	2://Prepear Write array befor write over ads
		//Standart Value
		//Type BOOL
		IF Lynus_Standards.GVL_Communicator.arrInterfaceInfoValueWriteTo[byReadWriteArrayNumber].sSymbolType = 'BOOL' AND TO_LWORD(Lynus_Standards.GVL_Communicator.arrInterfaceInfoValueWriteTo[byReadWriteArrayNumber].arrValue[1]) >= 0 AND TO_LWORD(Lynus_Standards.GVL_Communicator.arrInterfaceInfoValueWriteTo[byReadWriteArrayNumber].arrValue[1]) <= 1 THEN 
			arrBufferWrite_WriteAds[1] := STRING_TO_BYTE(Lynus_Standards.GVL_Communicator.arrInterfaceInfoValueWriteTo[byReadWriteArrayNumber].arrValue[1]); 
				bValueValid_WriteAds := TRUE;
					uiSizeToWrite_WriteAds := 1;
		END_IF
		//Type BYTE  	
		IF Lynus_Standards.GVL_Communicator.arrInterfaceInfoValueWriteTo[byReadWriteArrayNumber].sSymbolType = 'BYTE' AND TO_LWORD(Lynus_Standards.GVL_Communicator.arrInterfaceInfoValueWriteTo[byReadWriteArrayNumber].arrValue[1]) >= 0 AND TO_LWORD(Lynus_Standards.GVL_Communicator.arrInterfaceInfoValueWriteTo[byReadWriteArrayNumber].arrValue[1]) <= 255 THEN 
			arrBufferWrite_WriteAds[1] := STRING_TO_BYTE(Lynus_Standards.GVL_Communicator.arrInterfaceInfoValueWriteTo[byReadWriteArrayNumber].arrValue[1]); 
				bValueValid_WriteAds := TRUE;
					uiSizeToWrite_WriteAds := 1;
		END_IF
		//Type WORD
		IF Lynus_Standards.GVL_Communicator.arrInterfaceInfoValueWriteTo[byReadWriteArrayNumber].sSymbolType = 'WORD' AND TO_LWORD(Lynus_Standards.GVL_Communicator.arrInterfaceInfoValueWriteTo[byReadWriteArrayNumber].arrValue[1]) >= 0 AND TO_LWORD(Lynus_Standards.GVL_Communicator.arrInterfaceInfoValueWriteTo[byReadWriteArrayNumber].arrValue[1]) <= 65535 THEN 
			arrBufferWrite_WriteAds[2] := WORD_TO_BYTE(SHR(STRING_TO_WORD(Lynus_Standards.GVL_Communicator.arrInterfaceInfoValueWriteTo[byReadWriteArrayNumber].arrValue[1]),8) AND 16#FFFF);
			arrBufferWrite_WriteAds[1] := WORD_TO_BYTE(STRING_TO_WORD(Lynus_Standards.GVL_Communicator.arrInterfaceInfoValueWriteTo[byReadWriteArrayNumber].arrValue[1]) AND 16#FFFF); 
				bValueValid_WriteAds := TRUE;
					uiSizeToWrite_WriteAds := 2;
		END_IF
		//Type DWORD
		IF Lynus_Standards.GVL_Communicator.arrInterfaceInfoValueWriteTo[byReadWriteArrayNumber].sSymbolType = 'DWORD' AND TO_LWORD(Lynus_Standards.GVL_Communicator.arrInterfaceInfoValueWriteTo[byReadWriteArrayNumber].arrValue[1]) >= 0 AND TO_LWORD(Lynus_Standards.GVL_Communicator.arrInterfaceInfoValueWriteTo[byReadWriteArrayNumber].arrValue[1]) <= 4294967295 THEN 
			arrBufferWrite_WriteAds[4] := DWORD_TO_BYTE(SHR(STRING_TO_DWORD(Lynus_Standards.GVL_Communicator.arrInterfaceInfoValueWriteTo[byReadWriteArrayNumber].arrValue[1]),24) AND 16#FFFFFFFF);
			arrBufferWrite_WriteAds[3] := DWORD_TO_BYTE(SHR(STRING_TO_DWORD(Lynus_Standards.GVL_Communicator.arrInterfaceInfoValueWriteTo[byReadWriteArrayNumber].arrValue[1]),16) AND 16#FFFFFFFF);
			arrBufferWrite_WriteAds[2] := DWORD_TO_BYTE(SHR(STRING_TO_DWORD(Lynus_Standards.GVL_Communicator.arrInterfaceInfoValueWriteTo[byReadWriteArrayNumber].arrValue[1]),8) AND 16#FFFFFFFF);
			arrBufferWrite_WriteAds[1] := DWORD_TO_BYTE(STRING_TO_DWORD(Lynus_Standards.GVL_Communicator.arrInterfaceInfoValueWriteTo[byReadWriteArrayNumber].arrValue[1]) AND 16#FFFFFFFF); 
				bValueValid_WriteAds := TRUE;
					uiSizeToWrite_WriteAds := 4;
		END_IF
		//Type SINT
		IF Lynus_Standards.GVL_Communicator.arrInterfaceInfoValueWriteTo[byReadWriteArrayNumber].sSymbolType = 'SINT' AND TO_LINT(Lynus_Standards.GVL_Communicator.arrInterfaceInfoValueWriteTo[byReadWriteArrayNumber].arrValue[1]) >= -128 AND TO_LINT(Lynus_Standards.GVL_Communicator.arrInterfaceInfoValueWriteTo[byReadWriteArrayNumber].arrValue[1]) <= 127 THEN 
			arrBufferWrite_WriteAds[1] := SINT_TO_BYTE(STRING_TO_SINT(Lynus_Standards.GVL_Communicator.arrInterfaceInfoValueWriteTo[byReadWriteArrayNumber].arrValue[1])); 
				bValueValid_WriteAds := TRUE;
					uiSizeToWrite_WriteAds := 1;
		END_IF
		//Type USINT
		IF Lynus_Standards.GVL_Communicator.arrInterfaceInfoValueWriteTo[byReadWriteArrayNumber].sSymbolType = 'USINT' AND TO_LWORD(Lynus_Standards.GVL_Communicator.arrInterfaceInfoValueWriteTo[byReadWriteArrayNumber].arrValue[1]) >= 0 AND TO_LWORD(Lynus_Standards.GVL_Communicator.arrInterfaceInfoValueWriteTo[byReadWriteArrayNumber].arrValue[1]) <= 255 THEN 
			arrBufferWrite_WriteAds[1] := arrBufferWrite_WriteAds[1] := STRING_TO_USINT(Lynus_Standards.GVL_Communicator.arrInterfaceInfoValueWriteTo[byReadWriteArrayNumber].arrValue[1]); 
				bValueValid_WriteAds := TRUE;
					uiSizeToWrite_WriteAds := 1;
		END_IF
		//Type INT
		IF Lynus_Standards.GVL_Communicator.arrInterfaceInfoValueWriteTo[byReadWriteArrayNumber].sSymbolType = 'INT' AND TO_LINT(Lynus_Standards.GVL_Communicator.arrInterfaceInfoValueWriteTo[byReadWriteArrayNumber].arrValue[1]) >= -32768 AND TO_LINT(Lynus_Standards.GVL_Communicator.arrInterfaceInfoValueWriteTo[byReadWriteArrayNumber].arrValue[1]) <= 32767 THEN 
			arrBufferWrite_WriteAds[2] := UINT_TO_BYTE(SHR(INT_TO_UINT(STRING_TO_INT(Lynus_Standards.GVL_Communicator.arrInterfaceInfoValueWriteTo[byReadWriteArrayNumber].arrValue[1])),8) AND 16#FFFF);
			arrBufferWrite_WriteAds[1] := UINT_TO_BYTE(INT_TO_UINT(STRING_TO_INT(Lynus_Standards.GVL_Communicator.arrInterfaceInfoValueWriteTo[byReadWriteArrayNumber].arrValue[1])) AND 16#FFFF); 
				bValueValid_WriteAds := TRUE;
					uiSizeToWrite_WriteAds := 2;
		END_IF
		//Type UINT
		IF Lynus_Standards.GVL_Communicator.arrInterfaceInfoValueWriteTo[byReadWriteArrayNumber].sSymbolType = 'UINT' AND TO_LWORD(Lynus_Standards.GVL_Communicator.arrInterfaceInfoValueWriteTo[byReadWriteArrayNumber].arrValue[1]) >= 0 AND TO_LWORD(Lynus_Standards.GVL_Communicator.arrInterfaceInfoValueWriteTo[byReadWriteArrayNumber].arrValue[1]) <= 65535 THEN 
			arrBufferWrite_WriteAds[2] := UINT_TO_BYTE(SHR(STRING_TO_UINT(Lynus_Standards.GVL_Communicator.arrInterfaceInfoValueWriteTo[byReadWriteArrayNumber].arrValue[1]),8) AND 16#FFFF);
			arrBufferWrite_WriteAds[1] := UINT_TO_BYTE(STRING_TO_UINT(Lynus_Standards.GVL_Communicator.arrInterfaceInfoValueWriteTo[byReadWriteArrayNumber].arrValue[1]) AND 16#FFFF); 
				bValueValid_WriteAds := TRUE;
					uiSizeToWrite_WriteAds := 2;
		END_IF
		//Type DINT
		IF Lynus_Standards.GVL_Communicator.arrInterfaceInfoValueWriteTo[byReadWriteArrayNumber].sSymbolType = 'DINT' AND TO_LINT(Lynus_Standards.GVL_Communicator.arrInterfaceInfoValueWriteTo[byReadWriteArrayNumber].arrValue[1]) >= -2147483648 AND TO_LINT(Lynus_Standards.GVL_Communicator.arrInterfaceInfoValueWriteTo[byReadWriteArrayNumber].arrValue[1]) <= 2147483647 THEN 
			arrBufferWrite_WriteAds[4] := UDINT_TO_BYTE(SHR(DINT_TO_UDINT(STRING_TO_DINT(Lynus_Standards.GVL_Communicator.arrInterfaceInfoValueWriteTo[byReadWriteArrayNumber].arrValue[1])),24) AND 16#FFFFFFFF);
			arrBufferWrite_WriteAds[3] := UDINT_TO_BYTE(SHR(DINT_TO_UDINT(STRING_TO_DINT(Lynus_Standards.GVL_Communicator.arrInterfaceInfoValueWriteTo[byReadWriteArrayNumber].arrValue[1])),16) AND 16#FFFFFFFF);
			arrBufferWrite_WriteAds[2] := UDINT_TO_BYTE(SHR(DINT_TO_UDINT(STRING_TO_DINT(Lynus_Standards.GVL_Communicator.arrInterfaceInfoValueWriteTo[byReadWriteArrayNumber].arrValue[1])),8) AND 16#FFFFFFFF);
			arrBufferWrite_WriteAds[1] := UDINT_TO_BYTE(DINT_TO_UDINT(STRING_TO_DINT(Lynus_Standards.GVL_Communicator.arrInterfaceInfoValueWriteTo[byReadWriteArrayNumber].arrValue[1])) AND 16#FFFFFFF);
				bValueValid_WriteAds := TRUE;
					uiSizeToWrite_WriteAds := 4;
		END_IF
		//Type UDINT
		IF Lynus_Standards.GVL_Communicator.arrInterfaceInfoValueWriteTo[byReadWriteArrayNumber].sSymbolType = 'UDINT' AND TO_LWORD(Lynus_Standards.GVL_Communicator.arrInterfaceInfoValueWriteTo[byReadWriteArrayNumber].arrValue[1]) >= 0 AND TO_LWORD(Lynus_Standards.GVL_Communicator.arrInterfaceInfoValueWriteTo[byReadWriteArrayNumber].arrValue[1]) <= 4294967295 THEN 
			arrBufferWrite_WriteAds[4] := UDINT_TO_BYTE(SHR(STRING_TO_UDINT(Lynus_Standards.GVL_Communicator.arrInterfaceInfoValueWriteTo[byReadWriteArrayNumber].arrValue[1]),24) AND 16#FFFFFFFF);
			arrBufferWrite_WriteAds[3] := UDINT_TO_BYTE(SHR(STRING_TO_UDINT(Lynus_Standards.GVL_Communicator.arrInterfaceInfoValueWriteTo[byReadWriteArrayNumber].arrValue[1]),16) AND 16#FFFFFFFF);
			arrBufferWrite_WriteAds[2] := UDINT_TO_BYTE(SHR(STRING_TO_UDINT(Lynus_Standards.GVL_Communicator.arrInterfaceInfoValueWriteTo[byReadWriteArrayNumber].arrValue[1]),8) AND 16#FFFFFFFF);
			arrBufferWrite_WriteAds[1] := UDINT_TO_BYTE(STRING_TO_UDINT(Lynus_Standards.GVL_Communicator.arrInterfaceInfoValueWriteTo[byReadWriteArrayNumber].arrValue[1]) AND 16#FFFFFFFF); 
				bValueValid_WriteAds := TRUE;
					uiSizeToWrite_WriteAds := 4;
		END_IF
		//Type LINT
		IF Lynus_Standards.GVL_Communicator.arrInterfaceInfoValueWriteTo[byReadWriteArrayNumber].sSymbolType = 'LINT' AND TO_LINT(Lynus_Standards.GVL_Communicator.arrInterfaceInfoValueWriteTo[byReadWriteArrayNumber].arrValue[1]) >= -9223372036854775808 AND TO_LINT(Lynus_Standards.GVL_Communicator.arrInterfaceInfoValueWriteTo[byReadWriteArrayNumber].arrValue[1]) <= 9223372036854775807 THEN 
			arrBufferWrite_WriteAds[8] := ULINT_TO_BYTE(SHR(LINT_TO_ULINT(STRING_TO_LINT(Lynus_Standards.GVL_Communicator.arrInterfaceInfoValueWriteTo[byReadWriteArrayNumber].arrValue[1])),56) AND 16#FFFFFFFFFFFFFFFF);
			arrBufferWrite_WriteAds[7] := ULINT_TO_BYTE(SHR(LINT_TO_ULINT(STRING_TO_LINT(Lynus_Standards.GVL_Communicator.arrInterfaceInfoValueWriteTo[byReadWriteArrayNumber].arrValue[1])),48) AND 16#FFFFFFFFFFFFFFFF);
			arrBufferWrite_WriteAds[6] := ULINT_TO_BYTE(SHR(LINT_TO_ULINT(STRING_TO_LINT(Lynus_Standards.GVL_Communicator.arrInterfaceInfoValueWriteTo[byReadWriteArrayNumber].arrValue[1])),40) AND 16#FFFFFFFFFFFFFFFF);
			arrBufferWrite_WriteAds[5] := ULINT_TO_BYTE(SHR(LINT_TO_ULINT(STRING_TO_LINT(Lynus_Standards.GVL_Communicator.arrInterfaceInfoValueWriteTo[byReadWriteArrayNumber].arrValue[1])),32) AND 16#FFFFFFFFFFFFFFFF);
			arrBufferWrite_WriteAds[4] := ULINT_TO_BYTE(SHR(LINT_TO_ULINT(STRING_TO_LINT(Lynus_Standards.GVL_Communicator.arrInterfaceInfoValueWriteTo[byReadWriteArrayNumber].arrValue[1])),24) AND 16#FFFFFFFFFFFFFFFF);
			arrBufferWrite_WriteAds[3] := ULINT_TO_BYTE(SHR(LINT_TO_ULINT(STRING_TO_LINT(Lynus_Standards.GVL_Communicator.arrInterfaceInfoValueWriteTo[byReadWriteArrayNumber].arrValue[1])),16) AND 16#FFFFFFFFFFFFFFFF);
			arrBufferWrite_WriteAds[2] := ULINT_TO_BYTE(SHR(LINT_TO_ULINT(STRING_TO_LINT(Lynus_Standards.GVL_Communicator.arrInterfaceInfoValueWriteTo[byReadWriteArrayNumber].arrValue[1])),8) AND 16#FFFFFFFFFFFFFFFF);
			arrBufferWrite_WriteAds[1] := ULINT_TO_BYTE(LINT_TO_ULINT(STRING_TO_LINT(Lynus_Standards.GVL_Communicator.arrInterfaceInfoValueWriteTo[byReadWriteArrayNumber].arrValue[1])) AND 16#FFFFFFFFFFFFFFFF);
				bValueValid_WriteAds := TRUE;
					uiSizeToWrite_WriteAds := 8;
		END_IF
		//Type ULINT
		IF Lynus_Standards.GVL_Communicator.arrInterfaceInfoValueWriteTo[byReadWriteArrayNumber].sSymbolType = 'ULINT' AND TO_ULINT(Lynus_Standards.GVL_Communicator.arrInterfaceInfoValueWriteTo[byReadWriteArrayNumber].arrValue[1]) >= 0 AND TO_ULINT(Lynus_Standards.GVL_Communicator.arrInterfaceInfoValueWriteTo[byReadWriteArrayNumber].arrValue[1]) <= 18446744073709551615 THEN 
			arrBufferWrite_WriteAds[8] := ULINT_TO_BYTE(SHR(STRING_TO_ULINT(Lynus_Standards.GVL_Communicator.arrInterfaceInfoValueWriteTo[byReadWriteArrayNumber].arrValue[1]),56) AND 16#FFFFFFFFFFFFFFFF);
			arrBufferWrite_WriteAds[7] := ULINT_TO_BYTE(SHR(STRING_TO_ULINT(Lynus_Standards.GVL_Communicator.arrInterfaceInfoValueWriteTo[byReadWriteArrayNumber].arrValue[1]),48) AND 16#FFFFFFFFFFFFFFFF);
			arrBufferWrite_WriteAds[6] := ULINT_TO_BYTE(SHR(STRING_TO_ULINT(Lynus_Standards.GVL_Communicator.arrInterfaceInfoValueWriteTo[byReadWriteArrayNumber].arrValue[1]),40) AND 16#FFFFFFFFFFFFFFFF);
			arrBufferWrite_WriteAds[5] := ULINT_TO_BYTE(SHR(STRING_TO_ULINT(Lynus_Standards.GVL_Communicator.arrInterfaceInfoValueWriteTo[byReadWriteArrayNumber].arrValue[1]),32) AND 16#FFFFFFFFFFFFFFFF);
			arrBufferWrite_WriteAds[4] := ULINT_TO_BYTE(SHR(STRING_TO_ULINT(Lynus_Standards.GVL_Communicator.arrInterfaceInfoValueWriteTo[byReadWriteArrayNumber].arrValue[1]),24) AND 16#FFFFFFFFFFFFFFFF);
			arrBufferWrite_WriteAds[3] := ULINT_TO_BYTE(SHR(STRING_TO_ULINT(Lynus_Standards.GVL_Communicator.arrInterfaceInfoValueWriteTo[byReadWriteArrayNumber].arrValue[1]),16) AND 16#FFFFFFFFFFFFFFFF);
			arrBufferWrite_WriteAds[2] := ULINT_TO_BYTE(SHR(STRING_TO_ULINT(Lynus_Standards.GVL_Communicator.arrInterfaceInfoValueWriteTo[byReadWriteArrayNumber].arrValue[1]),8) AND 16#FFFFFFFFFFFFFFFF);
			arrBufferWrite_WriteAds[1] := ULINT_TO_BYTE(STRING_TO_ULINT(Lynus_Standards.GVL_Communicator.arrInterfaceInfoValueWriteTo[byReadWriteArrayNumber].arrValue[1]) AND 16#FFFFFFFFFFFFFFFF);
				bValueValid_WriteAds := TRUE;
					uiSizeToWrite_WriteAds := 8;
		END_IF
		//Type LWORD
		IF Lynus_Standards.GVL_Communicator.arrInterfaceInfoValueWriteTo[byReadWriteArrayNumber].sSymbolType = 'LWORD' AND TO_LWORD(Lynus_Standards.GVL_Communicator.arrInterfaceInfoValueWriteTo[byReadWriteArrayNumber].arrValue[1]) >= 0 AND TO_LWORD(Lynus_Standards.GVL_Communicator.arrInterfaceInfoValueWriteTo[byReadWriteArrayNumber].arrValue[1]) <= 18446744073709551615 THEN 
			arrBufferWrite_WriteAds[8] := LWORD_TO_BYTE(SHR(STRING_TO_LWORD(Lynus_Standards.GVL_Communicator.arrInterfaceInfoValueWriteTo[byReadWriteArrayNumber].arrValue[1]),56) AND 16#FFFFFFFFFFFFFFFF);
			arrBufferWrite_WriteAds[7] := LWORD_TO_BYTE(SHR(STRING_TO_LWORD(Lynus_Standards.GVL_Communicator.arrInterfaceInfoValueWriteTo[byReadWriteArrayNumber].arrValue[1]),48) AND 16#FFFFFFFFFFFFFFFF);
			arrBufferWrite_WriteAds[6] := LWORD_TO_BYTE(SHR(STRING_TO_LWORD(Lynus_Standards.GVL_Communicator.arrInterfaceInfoValueWriteTo[byReadWriteArrayNumber].arrValue[1]),40) AND 16#FFFFFFFFFFFFFFFF);
			arrBufferWrite_WriteAds[5] := LWORD_TO_BYTE(SHR(STRING_TO_LWORD(Lynus_Standards.GVL_Communicator.arrInterfaceInfoValueWriteTo[byReadWriteArrayNumber].arrValue[1]),32) AND 16#FFFFFFFFFFFFFFFF);
			arrBufferWrite_WriteAds[4] := LWORD_TO_BYTE(SHR(STRING_TO_LWORD(Lynus_Standards.GVL_Communicator.arrInterfaceInfoValueWriteTo[byReadWriteArrayNumber].arrValue[1]),24) AND 16#FFFFFFFFFFFFFFFF);
			arrBufferWrite_WriteAds[3] := LWORD_TO_BYTE(SHR(STRING_TO_LWORD(Lynus_Standards.GVL_Communicator.arrInterfaceInfoValueWriteTo[byReadWriteArrayNumber].arrValue[1]),16) AND 16#FFFFFFFFFFFFFFFF);
			arrBufferWrite_WriteAds[2] := LWORD_TO_BYTE(SHR(STRING_TO_LWORD(Lynus_Standards.GVL_Communicator.arrInterfaceInfoValueWriteTo[byReadWriteArrayNumber].arrValue[1]),8) AND 16#FFFFFFFFFFFFFFFF);
			arrBufferWrite_WriteAds[1] := LWORD_TO_BYTE(STRING_TO_LWORD(Lynus_Standards.GVL_Communicator.arrInterfaceInfoValueWriteTo[byReadWriteArrayNumber].arrValue[1]) AND 16#FFFFFFFFFFFFFFFF);
				bValueValid_WriteAds := TRUE;
					uiSizeToWrite_WriteAds := 8;
		END_IF
		//Type REAL
		IF Lynus_Standards.GVL_Communicator.arrInterfaceInfoValueWriteTo[byReadWriteArrayNumber].sSymbolType = 'REAL' AND LEN(Lynus_Standards.GVL_Communicator.arrInterfaceInfoValueWriteTo[byReadWriteArrayNumber].arrValue[1]) <= 30 AND TO_LREAL(Lynus_Standards.GVL_Communicator.arrInterfaceInfoValueWriteTo[byReadWriteArrayNumber].arrValue[1]) >= -3.40282326E+38 AND TO_LREAL(Lynus_Standards.GVL_Communicator.arrInterfaceInfoValueWriteTo[byReadWriteArrayNumber].arrValue[1]) <= 3.40282326E+38 THEN
			rRealValueCheckBeforWrite_WriteAds := STRING_TO_REAL(Lynus_Standards.GVL_Communicator.arrInterfaceInfoValueWriteTo[byReadWriteArrayNumber].arrValue[1]);
				IF IsFinite(F_REAL(rRealValueCheckBeforWrite_WriteAds)) THEN
					unConvertDWORD_TO_REAL_WriteAds.rValueFloat := STRING_TO_REAL(Lynus_Standards.GVL_Communicator.arrInterfaceInfoValueWriteTo[byReadWriteArrayNumber].arrValue[1]);
						arrBufferWrite_WriteAds[4] := UDINT_TO_BYTE((SHR(DWORD_TO_UDINT(unConvertDWORD_TO_REAL_WriteAds.dwRawValue),24) AND 16#FFFFFFFF));
						arrBufferWrite_WriteAds[3] := UDINT_TO_BYTE((SHR(DWORD_TO_UDINT(unConvertDWORD_TO_REAL_WriteAds.dwRawValue),16) AND 16#FFFFFFFF));
						arrBufferWrite_WriteAds[2] := UDINT_TO_BYTE((SHR(DWORD_TO_UDINT(unConvertDWORD_TO_REAL_WriteAds.dwRawValue),8) AND 16#FFFFFFFF));
						arrBufferWrite_WriteAds[1] := UDINT_TO_BYTE(DWORD_TO_UDINT(unConvertDWORD_TO_REAL_WriteAds.dwRawValue) AND 16#FFFFFFFF);
							bValueValid_WriteAds := TRUE;
								uiSizeToWrite_WriteAds := 4;
				END_IF					
		END_IF	
		//Type LREAL
		IF Lynus_Standards.GVL_Communicator.arrInterfaceInfoValueWriteTo[byReadWriteArrayNumber].sSymbolType = 'LREAL' AND LEN(Lynus_Standards.GVL_Communicator.arrInterfaceInfoValueWriteTo[byReadWriteArrayNumber].arrValue[1]) <= 30 AND TO_LREAL(Lynus_Standards.GVL_Communicator.arrInterfaceInfoValueWriteTo[byReadWriteArrayNumber].arrValue[1]) >= -1.7976931348623157E+307 AND TO_LREAL(Lynus_Standards.GVL_Communicator.arrInterfaceInfoValueWriteTo[byReadWriteArrayNumber].arrValue[1]) <= 1.7976931348623157E+307 THEN
			lrRealValueCheckBeforWrite_WriteAds := STRING_TO_LREAL(Lynus_Standards.GVL_Communicator.arrInterfaceInfoValueWriteTo[byReadWriteArrayNumber].arrValue[1]);
				IF IsFinite(F_LREAL(lrRealValueCheckBeforWrite_WriteAds)) THEN
					unConvertULINT_TO_LREAL_WriteAds.lrValueFloat := STRING_TO_LREAL(Lynus_Standards.GVL_Communicator.arrInterfaceInfoValueWriteTo[byReadWriteArrayNumber].arrValue[1]);
						arrBufferWrite_WriteAds[8] := LWORD_TO_BYTE((SHR(ULINT_TO_LWORD(unConvertULINT_TO_LREAL_WriteAds.uliRawValue),56) AND 16#FFFFFFFFFFFFFFFF));
						arrBufferWrite_WriteAds[7] := LWORD_TO_BYTE((SHR(ULINT_TO_LWORD(unConvertULINT_TO_LREAL_WriteAds.uliRawValue),48) AND 16#FFFFFFFFFFFFFFFF));
						arrBufferWrite_WriteAds[6] := LWORD_TO_BYTE((SHR(ULINT_TO_LWORD(unConvertULINT_TO_LREAL_WriteAds.uliRawValue),40) AND 16#FFFFFFFFFFFFFFFF));
						arrBufferWrite_WriteAds[5] := LWORD_TO_BYTE((SHR(ULINT_TO_LWORD(unConvertULINT_TO_LREAL_WriteAds.uliRawValue),32) AND 16#FFFFFFFFFFFFFFFF));
						arrBufferWrite_WriteAds[4] := LWORD_TO_BYTE((SHR(ULINT_TO_LWORD(unConvertULINT_TO_LREAL_WriteAds.uliRawValue),24) AND 16#FFFFFFFFFFFFFFFF));
						arrBufferWrite_WriteAds[3] := LWORD_TO_BYTE((SHR(ULINT_TO_LWORD(unConvertULINT_TO_LREAL_WriteAds.uliRawValue),16) AND 16#FFFFFFFFFFFFFFFF));
						arrBufferWrite_WriteAds[2] := LWORD_TO_BYTE((SHR(ULINT_TO_LWORD(unConvertULINT_TO_LREAL_WriteAds.uliRawValue),8) AND 16#FFFFFFFFFFFFFFFF));
						arrBufferWrite_WriteAds[1] := LWORD_TO_BYTE(ULINT_TO_LWORD(unConvertULINT_TO_LREAL_WriteAds.uliRawValue) AND 16#FFFFFFFFFFFFFFFF);
							bValueValid_WriteAds := TRUE;
								uiSizeToWrite_WriteAds := 8;
				END_IF
		END_IF
		//Type STRING(30)
		IF Lynus_Standards.GVL_Communicator.arrInterfaceInfoValueWriteTo[byReadWriteArrayNumber].sSymbolType = 'STRING(30)' AND LEN(Lynus_Standards.GVL_Communicator.arrInterfaceInfoValueWriteTo[byReadWriteArrayNumber].arrValue[1]) <= 30 AND FIND(Lynus_Standards.GVL_Communicator.arrInterfaceInfoValueWriteTo[byReadWriteArrayNumber].arrValue[1],'#EMPTY#') = 0 THEN 
			FOR byLPEncodeReceivedString_WriteAds := 1 TO 30 BY 1 DO 
				byCounterEncodeString_WriteAds := byCounterEncodeString_WriteAds + 1;
					byCounterEncodeString_WriteAds := LIMIT(1,byCounterEncodeString_WriteAds,30);
						arrBufferWrite_WriteAds[byCounterEncodeString_WriteAds] := F_ToASC(MID(Lynus_Standards.GVL_Communicator.arrInterfaceInfoValueWriteTo[byReadWriteArrayNumber].arrValue[1],1,byCounterEncodeString_WriteAds));
							bValueValid_WriteAds := TRUE;
								uiSizeToWrite_WriteAds := byCounterEncodeString_WriteAds + 1;
			END_FOR
		END_IF
		IF Lynus_Standards.GVL_Communicator.arrInterfaceInfoValueWriteTo[byReadWriteArrayNumber].sSymbolType = 'STRING(30)' AND LEN(Lynus_Standards.GVL_Communicator.arrInterfaceInfoValueWriteTo[byReadWriteArrayNumber].arrValue[1]) <= 30 AND FIND(Lynus_Standards.GVL_Communicator.arrInterfaceInfoValueWriteTo[byReadWriteArrayNumber].arrValue[1],'#EMPTY#') <> 0 THEN
			FOR byLPEncodeReceivedString_WriteAds := 1 TO 30 BY 1 DO 
				byCounterEncodeString_WriteAds := byCounterEncodeString_WriteAds + 1;
					byCounterEncodeString_WriteAds := LIMIT(1,byCounterEncodeString_WriteAds,30);
						arrBufferWrite_WriteAds[byCounterEncodeString_WriteAds] := F_ToASC('');
							bValueValid_WriteAds := TRUE;
								uiSizeToWrite_WriteAds := byCounterEncodeString_WriteAds + 1;
			END_FOR
		END_IF
		//Type TIME and TIME_OF_DAY
		IF ((Lynus_Standards.GVL_Communicator.arrInterfaceInfoValueWriteTo[byReadWriteArrayNumber].sSymbolType = 'TIME' OR Lynus_Standards.GVL_Communicator.arrInterfaceInfoValueWriteTo[byReadWriteArrayNumber].sSymbolType = 'TIME_OF_DAY') AND TO_LWORD(Lynus_Standards.GVL_Communicator.arrInterfaceInfoValueWriteTo[byReadWriteArrayNumber].arrValue[1]) >= 0 AND TO_LWORD(Lynus_Standards.GVL_Communicator.arrInterfaceInfoValueWriteTo[byReadWriteArrayNumber].arrValue[1]) <= 4294967295) THEN 
			arrBufferWrite_WriteAds[4] := UDINT_TO_BYTE(SHR(STRING_TO_UDINT(Lynus_Standards.GVL_Communicator.arrInterfaceInfoValueWriteTo[byReadWriteArrayNumber].arrValue[1]),24) AND 16#FFFFFFFF);
			arrBufferWrite_WriteAds[3] := UDINT_TO_BYTE(SHR(STRING_TO_UDINT(Lynus_Standards.GVL_Communicator.arrInterfaceInfoValueWriteTo[byReadWriteArrayNumber].arrValue[1]),16) AND 16#FFFFFFFF);
			arrBufferWrite_WriteAds[2] := UDINT_TO_BYTE(SHR(STRING_TO_UDINT(Lynus_Standards.GVL_Communicator.arrInterfaceInfoValueWriteTo[byReadWriteArrayNumber].arrValue[1]),8) AND 16#FFFFFFFF);
			arrBufferWrite_WriteAds[1] := UDINT_TO_BYTE(STRING_TO_UDINT(Lynus_Standards.GVL_Communicator.arrInterfaceInfoValueWriteTo[byReadWriteArrayNumber].arrValue[1]) AND 16#FFFFFFFF); 
				bValueValid_WriteAds := TRUE;
					uiSizeToWrite_WriteAds := 4;
		END_IF
		//Type DATE and DATE_AND_TIME
		IF ((Lynus_Standards.GVL_Communicator.arrInterfaceInfoValueWriteTo[byReadWriteArrayNumber].sSymbolType = 'DATE' OR Lynus_Standards.GVL_Communicator.arrInterfaceInfoValueWriteTo[byReadWriteArrayNumber].sSymbolType = 'DATE_AND_TIME') AND TO_LWORD(Lynus_Standards.GVL_Communicator.arrInterfaceInfoValueWriteTo[byReadWriteArrayNumber].arrValue[1]) >= 0 AND TO_LWORD(Lynus_Standards.GVL_Communicator.arrInterfaceInfoValueWriteTo[byReadWriteArrayNumber].arrValue[1]) <= 4294967295000) THEN 
			uliDate_WriteAds := STRING_TO_ULINT(Lynus_Standards.GVL_Communicator.arrInterfaceInfoValueWriteTo[byReadWriteArrayNumber].arrValue[1]);
				udiDate_WriteAds := ULINT_TO_UDINT(uliDate_WriteAds / 1000);	
					arrBufferWrite_WriteAds[4] := UDINT_TO_BYTE(SHR(udiDate_WriteAds,24) AND 16#FFFFFFFF);
					arrBufferWrite_WriteAds[3] := UDINT_TO_BYTE(SHR(udiDate_WriteAds,16) AND 16#FFFFFFFF);
					arrBufferWrite_WriteAds[2] := UDINT_TO_BYTE(SHR(udiDate_WriteAds,8) AND 16#FFFFFFFF);
					arrBufferWrite_WriteAds[1] := UDINT_TO_BYTE(udiDate_WriteAds AND 16#FFFFFFFF); 
						bValueValid_WriteAds := TRUE;
							uiSizeToWrite_WriteAds := 4;
		END_IF
			//Array with Standart Value
			//Type BOOL
			IF Lynus_Standards.GVL_Communicator.arrInterfaceInfoValueWriteTo[byReadWriteArrayNumber].uiSizeArray <= Lynus_Standards.Constants_Communicator.bySizeOfValueArray AND FIND(Lynus_Standards.GVL_Communicator.arrInterfaceInfoValueWriteTo[byReadWriteArrayNumber].sSymbolType,'OF BOOL') <> 0 THEN
				FOR uiLPWriteValueFromArray_WriteAds := 1 TO Lynus_Standards.GVL_Communicator.arrInterfaceInfoValueWriteTo[byReadWriteArrayNumber].uiSizeArray BY 1 DO
					IF TO_LWORD(Lynus_Standards.GVL_Communicator.arrInterfaceInfoValueWriteTo[byReadWriteArrayNumber].arrValue[uiLPWriteValueFromArray_WriteAds]) >= 0 AND TO_LWORD(Lynus_Standards.GVL_Communicator.arrInterfaceInfoValueWriteTo[byReadWriteArrayNumber].arrValue[uiLPWriteValueFromArray_WriteAds]) <= 1 THEN   
						arrBufferWrite_WriteAds[uiLPWriteValueFromArray_WriteAds] := STRING_TO_BYTE(Lynus_Standards.GVL_Communicator.arrInterfaceInfoValueWriteTo[byReadWriteArrayNumber].arrValue[uiLPWriteValueFromArray_WriteAds]); 
							uiSizeToWrite_WriteAds := 1 * Lynus_Standards.GVL_Communicator.arrInterfaceInfoValueWriteTo[byReadWriteArrayNumber].uiSizeArray;
								byCounterReceivedValueOK_WriteAds := byCounterReceivedValueOK_WriteAds + 1;
									byCounterReceivedValueOK_WriteAds := LIMIT(0,byCounterReceivedValueOK_WriteAds,Lynus_Standards.Constants_Communicator.bySizeOfValueArray);
										IF byCounterReceivedValueOK_WriteAds >= Lynus_Standards.GVL_Communicator.arrInterfaceInfoValueWriteTo[byReadWriteArrayNumber].uiSizeArray THEN bValueValid_WriteAds := TRUE; END_IF 
					END_IF
				END_FOR
			END_IF
			//Type BYTE
			IF Lynus_Standards.GVL_Communicator.arrInterfaceInfoValueWriteTo[byReadWriteArrayNumber].uiSizeArray <= Lynus_Standards.Constants_Communicator.bySizeOfValueArray AND FIND(Lynus_Standards.GVL_Communicator.arrInterfaceInfoValueWriteTo[byReadWriteArrayNumber].sSymbolType,'OF BYTE') <> 0 THEN
				FOR uiLPWriteValueFromArray_WriteAds := 1 TO Lynus_Standards.GVL_Communicator.arrInterfaceInfoValueWriteTo[byReadWriteArrayNumber].uiSizeArray BY 1 DO   
					IF TO_LWORD(Lynus_Standards.GVL_Communicator.arrInterfaceInfoValueWriteTo[byReadWriteArrayNumber].arrValue[uiLPWriteValueFromArray_WriteAds]) >= 0 AND TO_LWORD(Lynus_Standards.GVL_Communicator.arrInterfaceInfoValueWriteTo[byReadWriteArrayNumber].arrValue[uiLPWriteValueFromArray_WriteAds]) <= 255 THEN 
						arrBufferWrite_WriteAds[uiLPWriteValueFromArray_WriteAds] := STRING_TO_BYTE(Lynus_Standards.GVL_Communicator.arrInterfaceInfoValueWriteTo[byReadWriteArrayNumber].arrValue[uiLPWriteValueFromArray_WriteAds]); 
							uiSizeToWrite_WriteAds := 1 * Lynus_Standards.GVL_Communicator.arrInterfaceInfoValueWriteTo[byReadWriteArrayNumber].uiSizeArray;
								byCounterReceivedValueOK_WriteAds := byCounterReceivedValueOK_WriteAds + 1;
									byCounterReceivedValueOK_WriteAds := LIMIT(0,byCounterReceivedValueOK_WriteAds,Lynus_Standards.Constants_Communicator.bySizeOfValueArray);
										IF byCounterReceivedValueOK_WriteAds >= Lynus_Standards.GVL_Communicator.arrInterfaceInfoValueWriteTo[byReadWriteArrayNumber].uiSizeArray THEN bValueValid_WriteAds := TRUE; END_IF  
					END_IF
				END_FOR
			END_IF
			//Type WORD
			IF Lynus_Standards.GVL_Communicator.arrInterfaceInfoValueWriteTo[byReadWriteArrayNumber].uiSizeArray <= Lynus_Standards.Constants_Communicator.bySizeOfValueArray AND FIND(Lynus_Standards.GVL_Communicator.arrInterfaceInfoValueWriteTo[byReadWriteArrayNumber].sSymbolType,'OF WORD') <> 0 THEN
				FOR uiLPWriteValueFromArray_WriteAds := 1 TO Lynus_Standards.GVL_Communicator.arrInterfaceInfoValueWriteTo[byReadWriteArrayNumber].uiSizeArray BY 1 DO  
					IF TO_LWORD(Lynus_Standards.GVL_Communicator.arrInterfaceInfoValueWriteTo[byReadWriteArrayNumber].arrValue[uiLPWriteValueFromArray_WriteAds]) >= 0 AND TO_LWORD(Lynus_Standards.GVL_Communicator.arrInterfaceInfoValueWriteTo[byReadWriteArrayNumber].arrValue[uiLPWriteValueFromArray_WriteAds]) <= 65535 THEN  
						arrCounterWriteValueInArray_WriteAds[1] := LIMIT(1,arrCounterWriteValueInArray_WriteAds[1],2000); arrCounterWriteValueInArray_WriteAds[2] := LIMIT(2,arrCounterWriteValueInArray_WriteAds[2],2000);	
							arrBufferWrite_WriteAds[arrCounterWriteValueInArray_WriteAds[2]] := WORD_TO_BYTE(SHR(STRING_TO_WORD(Lynus_Standards.GVL_Communicator.arrInterfaceInfoValueWriteTo[byReadWriteArrayNumber].arrValue[uiLPWriteValueFromArray_WriteAds]),8) AND 16#FFFF);
							arrBufferWrite_WriteAds[arrCounterWriteValueInArray_WriteAds[1]] := WORD_TO_BYTE(STRING_TO_WORD(Lynus_Standards.GVL_Communicator.arrInterfaceInfoValueWriteTo[byReadWriteArrayNumber].arrValue[uiLPWriteValueFromArray_WriteAds]) AND 16#FFFF); 
						arrCounterWriteValueInArray_WriteAds[1] := arrCounterWriteValueInArray_WriteAds[1] + 2; arrCounterWriteValueInArray_WriteAds[2] := arrCounterWriteValueInArray_WriteAds[2] + 2;
							uiSizeToWrite_WriteAds := 2 * Lynus_Standards.GVL_Communicator.arrInterfaceInfoValueWriteTo[byReadWriteArrayNumber].uiSizeArray;
								byCounterReceivedValueOK_WriteAds := byCounterReceivedValueOK_WriteAds + 1;
									byCounterReceivedValueOK_WriteAds := LIMIT(0,byCounterReceivedValueOK_WriteAds,Lynus_Standards.Constants_Communicator.bySizeOfValueArray);
										IF byCounterReceivedValueOK_WriteAds >= Lynus_Standards.GVL_Communicator.arrInterfaceInfoValueWriteTo[byReadWriteArrayNumber].uiSizeArray THEN bValueValid_WriteAds := TRUE; END_IF  
					END_IF
				END_FOR
			END_IF
			//Type DWORD
			IF Lynus_Standards.GVL_Communicator.arrInterfaceInfoValueWriteTo[byReadWriteArrayNumber].uiSizeArray <= Lynus_Standards.Constants_Communicator.bySizeOfValueArray AND FIND(Lynus_Standards.GVL_Communicator.arrInterfaceInfoValueWriteTo[byReadWriteArrayNumber].sSymbolType,'OF DWORD') <> 0 THEN
				FOR uiLPWriteValueFromArray_WriteAds := 1 TO Lynus_Standards.GVL_Communicator.arrInterfaceInfoValueWriteTo[byReadWriteArrayNumber].uiSizeArray BY 1 DO 
					IF TO_LWORD(Lynus_Standards.GVL_Communicator.arrInterfaceInfoValueWriteTo[byReadWriteArrayNumber].arrValue[uiLPWriteValueFromArray_WriteAds]) >= 0 AND TO_LWORD(Lynus_Standards.GVL_Communicator.arrInterfaceInfoValueWriteTo[byReadWriteArrayNumber].arrValue[uiLPWriteValueFromArray_WriteAds]) <= 4294967295 THEN   
						arrCounterWriteValueInArray_WriteAds[1] := LIMIT(1,arrCounterWriteValueInArray_WriteAds[1],2000); arrCounterWriteValueInArray_WriteAds[2] := LIMIT(2,arrCounterWriteValueInArray_WriteAds[2],2000);
							arrCounterWriteValueInArray_WriteAds[3] := LIMIT(3,arrCounterWriteValueInArray_WriteAds[3],2000); arrCounterWriteValueInArray_WriteAds[4] := LIMIT(4,arrCounterWriteValueInArray_WriteAds[4],2000);	
								arrBufferWrite_WriteAds[arrCounterWriteValueInArray_WriteAds[4]] := DWORD_TO_BYTE(SHR(STRING_TO_DWORD(Lynus_Standards.GVL_Communicator.arrInterfaceInfoValueWriteTo[byReadWriteArrayNumber].arrValue[uiLPWriteValueFromArray_WriteAds]),24) AND 16#FFFFFFFF);
								arrBufferWrite_WriteAds[arrCounterWriteValueInArray_WriteAds[3]] := DWORD_TO_BYTE(SHR(STRING_TO_DWORD(Lynus_Standards.GVL_Communicator.arrInterfaceInfoValueWriteTo[byReadWriteArrayNumber].arrValue[uiLPWriteValueFromArray_WriteAds]),16) AND 16#FFFFFFFF);
								arrBufferWrite_WriteAds[arrCounterWriteValueInArray_WriteAds[2]] := DWORD_TO_BYTE(SHR(STRING_TO_DWORD(Lynus_Standards.GVL_Communicator.arrInterfaceInfoValueWriteTo[byReadWriteArrayNumber].arrValue[uiLPWriteValueFromArray_WriteAds]),8) AND 16#FFFFFFFF);
								arrBufferWrite_WriteAds[arrCounterWriteValueInArray_WriteAds[1]] := DWORD_TO_BYTE(STRING_TO_DWORD(Lynus_Standards.GVL_Communicator.arrInterfaceInfoValueWriteTo[byReadWriteArrayNumber].arrValue[uiLPWriteValueFromArray_WriteAds]) AND 16#FFFFFFFF); 
						arrCounterWriteValueInArray_WriteAds[1] := arrCounterWriteValueInArray_WriteAds[1] + 4; arrCounterWriteValueInArray_WriteAds[2] := arrCounterWriteValueInArray_WriteAds[2] + 4;
							arrCounterWriteValueInArray_WriteAds[3] := arrCounterWriteValueInArray_WriteAds[3] + 4; arrCounterWriteValueInArray_WriteAds[4] := arrCounterWriteValueInArray_WriteAds[4] + 4;
								uiSizeToWrite_WriteAds := 4 * Lynus_Standards.GVL_Communicator.arrInterfaceInfoValueWriteTo[byReadWriteArrayNumber].uiSizeArray;	
									byCounterReceivedValueOK_WriteAds := byCounterReceivedValueOK_WriteAds + 1;
										byCounterReceivedValueOK_WriteAds := LIMIT(0,byCounterReceivedValueOK_WriteAds,Lynus_Standards.Constants_Communicator.bySizeOfValueArray);
											IF byCounterReceivedValueOK_WriteAds >= Lynus_Standards.GVL_Communicator.arrInterfaceInfoValueWriteTo[byReadWriteArrayNumber].uiSizeArray THEN bValueValid_WriteAds := TRUE; END_IF  
					END_IF
				END_FOR
			END_IF
			//Type SINT
			IF Lynus_Standards.GVL_Communicator.arrInterfaceInfoValueWriteTo[byReadWriteArrayNumber].uiSizeArray <= Lynus_Standards.Constants_Communicator.bySizeOfValueArray AND FIND(Lynus_Standards.GVL_Communicator.arrInterfaceInfoValueWriteTo[byReadWriteArrayNumber].sSymbolType,'OF USINT') <> 0 THEN
				FOR uiLPWriteValueFromArray_WriteAds := 1 TO Lynus_Standards.GVL_Communicator.arrInterfaceInfoValueWriteTo[byReadWriteArrayNumber].uiSizeArray BY 1 DO   
					IF TO_LINT(Lynus_Standards.GVL_Communicator.arrInterfaceInfoValueWriteTo[byReadWriteArrayNumber].arrValue[uiLPWriteValueFromArray_WriteAds]) >= -128 AND TO_LINT(Lynus_Standards.GVL_Communicator.arrInterfaceInfoValueWriteTo[byReadWriteArrayNumber].arrValue[uiLPWriteValueFromArray_WriteAds]) <= 127 THEN 
						arrBufferWrite_WriteAds[uiLPWriteValueFromArray_WriteAds] := SINT_TO_BYTE(STRING_TO_SINT(Lynus_Standards.GVL_Communicator.arrInterfaceInfoValueWriteTo[byReadWriteArrayNumber].arrValue[uiLPWriteValueFromArray_WriteAds])); 
							uiSizeToWrite_WriteAds := 1 * Lynus_Standards.GVL_Communicator.arrInterfaceInfoValueWriteTo[byReadWriteArrayNumber].uiSizeArray;
								byCounterReceivedValueOK_WriteAds := byCounterReceivedValueOK_WriteAds + 1;
									byCounterReceivedValueOK_WriteAds := LIMIT(0,byCounterReceivedValueOK_WriteAds,Lynus_Standards.Constants_Communicator.bySizeOfValueArray);
										IF byCounterReceivedValueOK_WriteAds >= Lynus_Standards.GVL_Communicator.arrInterfaceInfoValueWriteTo[byReadWriteArrayNumber].uiSizeArray THEN bValueValid_WriteAds := TRUE; END_IF  
					END_IF
				END_FOR
			END_IF
			//Type USINT
			IF Lynus_Standards.GVL_Communicator.arrInterfaceInfoValueWriteTo[byReadWriteArrayNumber].uiSizeArray <= Lynus_Standards.Constants_Communicator.bySizeOfValueArray AND FIND(Lynus_Standards.GVL_Communicator.arrInterfaceInfoValueWriteTo[byReadWriteArrayNumber].sSymbolType,'OF USINT') <> 0 THEN
				FOR uiLPWriteValueFromArray_WriteAds := 1 TO Lynus_Standards.GVL_Communicator.arrInterfaceInfoValueWriteTo[byReadWriteArrayNumber].uiSizeArray BY 1 DO   
					IF TO_LWORD(Lynus_Standards.GVL_Communicator.arrInterfaceInfoValueWriteTo[byReadWriteArrayNumber].arrValue[uiLPWriteValueFromArray_WriteAds]) >= 0 AND TO_LWORD(Lynus_Standards.GVL_Communicator.arrInterfaceInfoValueWriteTo[byReadWriteArrayNumber].arrValue[uiLPWriteValueFromArray_WriteAds]) <= 255 THEN 
						arrBufferWrite_WriteAds[uiLPWriteValueFromArray_WriteAds] := STRING_TO_USINT(Lynus_Standards.GVL_Communicator.arrInterfaceInfoValueWriteTo[byReadWriteArrayNumber].arrValue[uiLPWriteValueFromArray_WriteAds]); 
							uiSizeToWrite_WriteAds := 1 * Lynus_Standards.GVL_Communicator.arrInterfaceInfoValueWriteTo[byReadWriteArrayNumber].uiSizeArray;
								byCounterReceivedValueOK_WriteAds := byCounterReceivedValueOK_WriteAds + 1;
									byCounterReceivedValueOK_WriteAds := LIMIT(0,byCounterReceivedValueOK_WriteAds,Lynus_Standards.Constants_Communicator.bySizeOfValueArray);
										IF byCounterReceivedValueOK_WriteAds >= Lynus_Standards.GVL_Communicator.arrInterfaceInfoValueWriteTo[byReadWriteArrayNumber].uiSizeArray THEN bValueValid_WriteAds := TRUE; END_IF  
					END_IF
				END_FOR
			END_IF
			//Type INT
			IF Lynus_Standards.GVL_Communicator.arrInterfaceInfoValueWriteTo[byReadWriteArrayNumber].uiSizeArray <= Lynus_Standards.Constants_Communicator.bySizeOfValueArray AND FIND(Lynus_Standards.GVL_Communicator.arrInterfaceInfoValueWriteTo[byReadWriteArrayNumber].sSymbolType,'OF INT') <> 0 THEN
				FOR uiLPWriteValueFromArray_WriteAds := 1 TO Lynus_Standards.GVL_Communicator.arrInterfaceInfoValueWriteTo[byReadWriteArrayNumber].uiSizeArray BY 1 DO   
					IF TO_LINT(Lynus_Standards.GVL_Communicator.arrInterfaceInfoValueWriteTo[byReadWriteArrayNumber].arrValue[uiLPWriteValueFromArray_WriteAds]) >= -32768 AND TO_LINT(Lynus_Standards.GVL_Communicator.arrInterfaceInfoValueWriteTo[byReadWriteArrayNumber].arrValue[uiLPWriteValueFromArray_WriteAds]) <= 32767 THEN 
						arrCounterWriteValueInArray_WriteAds[1] := LIMIT(1,arrCounterWriteValueInArray_WriteAds[1],2000); arrCounterWriteValueInArray_WriteAds[2] := LIMIT(2,arrCounterWriteValueInArray_WriteAds[2],2000);	
							arrBufferWrite_WriteAds[arrCounterWriteValueInArray_WriteAds[2]] := UINT_TO_BYTE(SHR(INT_TO_UINT(STRING_TO_INT(Lynus_Standards.GVL_Communicator.arrInterfaceInfoValueWriteTo[byReadWriteArrayNumber].arrValue[uiLPWriteValueFromArray_WriteAds])),8) AND 16#FFFF);
							arrBufferWrite_WriteAds[arrCounterWriteValueInArray_WriteAds[1]] := UINT_TO_BYTE(INT_TO_UINT(STRING_TO_INT(Lynus_Standards.GVL_Communicator.arrInterfaceInfoValueWriteTo[byReadWriteArrayNumber].arrValue[uiLPWriteValueFromArray_WriteAds])) AND 16#FFFF); 
						arrCounterWriteValueInArray_WriteAds[1] := arrCounterWriteValueInArray_WriteAds[1] + 2; arrCounterWriteValueInArray_WriteAds[2] := arrCounterWriteValueInArray_WriteAds[2] + 2;
							uiSizeToWrite_WriteAds := 2 * Lynus_Standards.GVL_Communicator.arrInterfaceInfoValueWriteTo[byReadWriteArrayNumber].uiSizeArray;
								byCounterReceivedValueOK_WriteAds := byCounterReceivedValueOK_WriteAds + 1;
									byCounterReceivedValueOK_WriteAds := LIMIT(0,byCounterReceivedValueOK_WriteAds,Lynus_Standards.Constants_Communicator.bySizeOfValueArray);
										IF byCounterReceivedValueOK_WriteAds >= Lynus_Standards.GVL_Communicator.arrInterfaceInfoValueWriteTo[byReadWriteArrayNumber].uiSizeArray THEN bValueValid_WriteAds := TRUE; END_IF  
					END_IF
				END_FOR
			END_IF
			//Type UINT
			IF Lynus_Standards.GVL_Communicator.arrInterfaceInfoValueWriteTo[byReadWriteArrayNumber].uiSizeArray <= Lynus_Standards.Constants_Communicator.bySizeOfValueArray AND FIND(Lynus_Standards.GVL_Communicator.arrInterfaceInfoValueWriteTo[byReadWriteArrayNumber].sSymbolType,'OF UINT') <> 0 THEN
				FOR uiLPWriteValueFromArray_WriteAds := 1 TO Lynus_Standards.GVL_Communicator.arrInterfaceInfoValueWriteTo[byReadWriteArrayNumber].uiSizeArray BY 1 DO  
					IF TO_LWORD(Lynus_Standards.GVL_Communicator.arrInterfaceInfoValueWriteTo[byReadWriteArrayNumber].arrValue[uiLPWriteValueFromArray_WriteAds]) >= 0 AND TO_LWORD(Lynus_Standards.GVL_Communicator.arrInterfaceInfoValueWriteTo[byReadWriteArrayNumber].arrValue[uiLPWriteValueFromArray_WriteAds]) <= 65535 THEN  
						arrCounterWriteValueInArray_WriteAds[1] := LIMIT(1,arrCounterWriteValueInArray_WriteAds[1],2000); arrCounterWriteValueInArray_WriteAds[2] := LIMIT(2,arrCounterWriteValueInArray_WriteAds[2],2000);	
							arrBufferWrite_WriteAds[arrCounterWriteValueInArray_WriteAds[2]] := UINT_TO_BYTE(SHR(STRING_TO_UINT(Lynus_Standards.GVL_Communicator.arrInterfaceInfoValueWriteTo[byReadWriteArrayNumber].arrValue[uiLPWriteValueFromArray_WriteAds]),8) AND 16#FFFF);
							arrBufferWrite_WriteAds[arrCounterWriteValueInArray_WriteAds[1]] := UINT_TO_BYTE(STRING_TO_UINT(Lynus_Standards.GVL_Communicator.arrInterfaceInfoValueWriteTo[byReadWriteArrayNumber].arrValue[uiLPWriteValueFromArray_WriteAds]) AND 16#FFFF);  
						arrCounterWriteValueInArray_WriteAds[1] := arrCounterWriteValueInArray_WriteAds[1] + 2; arrCounterWriteValueInArray_WriteAds[2] := arrCounterWriteValueInArray_WriteAds[2] + 2;
							uiSizeToWrite_WriteAds := 2 * Lynus_Standards.GVL_Communicator.arrInterfaceInfoValueWriteTo[byReadWriteArrayNumber].uiSizeArray;
								byCounterReceivedValueOK_WriteAds := byCounterReceivedValueOK_WriteAds + 1;
									byCounterReceivedValueOK_WriteAds := LIMIT(0,byCounterReceivedValueOK_WriteAds,Lynus_Standards.Constants_Communicator.bySizeOfValueArray);
										IF byCounterReceivedValueOK_WriteAds >= Lynus_Standards.GVL_Communicator.arrInterfaceInfoValueWriteTo[byReadWriteArrayNumber].uiSizeArray THEN bValueValid_WriteAds := TRUE; END_IF  
					END_IF
				END_FOR
			END_IF
			//Type DINT
			IF Lynus_Standards.GVL_Communicator.arrInterfaceInfoValueWriteTo[byReadWriteArrayNumber].uiSizeArray <= Lynus_Standards.Constants_Communicator.bySizeOfValueArray AND FIND(Lynus_Standards.GVL_Communicator.arrInterfaceInfoValueWriteTo[byReadWriteArrayNumber].sSymbolType,'OF DINT') <> 0 THEN
				FOR uiLPWriteValueFromArray_WriteAds := 1 TO Lynus_Standards.GVL_Communicator.arrInterfaceInfoValueWriteTo[byReadWriteArrayNumber].uiSizeArray BY 1 DO 
					IF TO_LINT(Lynus_Standards.GVL_Communicator.arrInterfaceInfoValueWriteTo[byReadWriteArrayNumber].arrValue[uiLPWriteValueFromArray_WriteAds]) >= -2147483648 AND TO_LINT(Lynus_Standards.GVL_Communicator.arrInterfaceInfoValueWriteTo[byReadWriteArrayNumber].arrValue[uiLPWriteValueFromArray_WriteAds]) <= 2147483647 THEN   
						arrCounterWriteValueInArray_WriteAds[1] := LIMIT(1,arrCounterWriteValueInArray_WriteAds[1],2000); arrCounterWriteValueInArray_WriteAds[2] := LIMIT(2,arrCounterWriteValueInArray_WriteAds[2],2000);
							arrCounterWriteValueInArray_WriteAds[3] := LIMIT(3,arrCounterWriteValueInArray_WriteAds[3],2000); arrCounterWriteValueInArray_WriteAds[4] := LIMIT(4,arrCounterWriteValueInArray_WriteAds[4],2000);	
								arrBufferWrite_WriteAds[arrCounterWriteValueInArray_WriteAds[4]] := UDINT_TO_BYTE(SHR(DINT_TO_UDINT(STRING_TO_DINT(Lynus_Standards.GVL_Communicator.arrInterfaceInfoValueWriteTo[byReadWriteArrayNumber].arrValue[uiLPWriteValueFromArray_WriteAds])),24) AND 16#FFFFFFFF);
								arrBufferWrite_WriteAds[arrCounterWriteValueInArray_WriteAds[3]] := UDINT_TO_BYTE(SHR(DINT_TO_UDINT(STRING_TO_DINT(Lynus_Standards.GVL_Communicator.arrInterfaceInfoValueWriteTo[byReadWriteArrayNumber].arrValue[uiLPWriteValueFromArray_WriteAds])),16) AND 16#FFFFFFFF);
								arrBufferWrite_WriteAds[arrCounterWriteValueInArray_WriteAds[2]] := UDINT_TO_BYTE(SHR(DINT_TO_UDINT(STRING_TO_DINT(Lynus_Standards.GVL_Communicator.arrInterfaceInfoValueWriteTo[byReadWriteArrayNumber].arrValue[uiLPWriteValueFromArray_WriteAds])),8) AND 16#FFFFFFFF);
								arrBufferWrite_WriteAds[arrCounterWriteValueInArray_WriteAds[1]] := UDINT_TO_BYTE(DINT_TO_UDINT(STRING_TO_DINT(Lynus_Standards.GVL_Communicator.arrInterfaceInfoValueWriteTo[byReadWriteArrayNumber].arrValue[uiLPWriteValueFromArray_WriteAds])) AND 16#FFFFFFF); 
						arrCounterWriteValueInArray_WriteAds[1] := arrCounterWriteValueInArray_WriteAds[1] + 4; arrCounterWriteValueInArray_WriteAds[2] := arrCounterWriteValueInArray_WriteAds[2] + 4;
							arrCounterWriteValueInArray_WriteAds[3] := arrCounterWriteValueInArray_WriteAds[3] + 4; arrCounterWriteValueInArray_WriteAds[4] := arrCounterWriteValueInArray_WriteAds[4] + 4;
								uiSizeToWrite_WriteAds := 4 * Lynus_Standards.GVL_Communicator.arrInterfaceInfoValueWriteTo[byReadWriteArrayNumber].uiSizeArray;	
									byCounterReceivedValueOK_WriteAds := byCounterReceivedValueOK_WriteAds + 1;
										byCounterReceivedValueOK_WriteAds := LIMIT(0,byCounterReceivedValueOK_WriteAds,Lynus_Standards.Constants_Communicator.bySizeOfValueArray);
											IF byCounterReceivedValueOK_WriteAds >= Lynus_Standards.GVL_Communicator.arrInterfaceInfoValueWriteTo[byReadWriteArrayNumber].uiSizeArray THEN bValueValid_WriteAds := TRUE; END_IF  
					END_IF
				END_FOR
			END_IF
			//Type UDINT
			IF Lynus_Standards.GVL_Communicator.arrInterfaceInfoValueWriteTo[byReadWriteArrayNumber].uiSizeArray <= Lynus_Standards.Constants_Communicator.bySizeOfValueArray AND FIND(Lynus_Standards.GVL_Communicator.arrInterfaceInfoValueWriteTo[byReadWriteArrayNumber].sSymbolType,'OF UDINT') <> 0 THEN
				FOR uiLPWriteValueFromArray_WriteAds := 1 TO Lynus_Standards.GVL_Communicator.arrInterfaceInfoValueWriteTo[byReadWriteArrayNumber].uiSizeArray BY 1 DO 
					IF TO_LWORD(Lynus_Standards.GVL_Communicator.arrInterfaceInfoValueWriteTo[byReadWriteArrayNumber].arrValue[uiLPWriteValueFromArray_WriteAds]) >= 0 AND TO_LWORD(Lynus_Standards.GVL_Communicator.arrInterfaceInfoValueWriteTo[byReadWriteArrayNumber].arrValue[uiLPWriteValueFromArray_WriteAds]) <= 4294967295 THEN   
						arrCounterWriteValueInArray_WriteAds[1] := LIMIT(1,arrCounterWriteValueInArray_WriteAds[1],2000); arrCounterWriteValueInArray_WriteAds[2] := LIMIT(2,arrCounterWriteValueInArray_WriteAds[2],2000);
							arrCounterWriteValueInArray_WriteAds[3] := LIMIT(3,arrCounterWriteValueInArray_WriteAds[3],2000); arrCounterWriteValueInArray_WriteAds[4] := LIMIT(4,arrCounterWriteValueInArray_WriteAds[4],2000);	
								arrBufferWrite_WriteAds[arrCounterWriteValueInArray_WriteAds[4]] := UDINT_TO_BYTE(SHR(STRING_TO_UDINT(Lynus_Standards.GVL_Communicator.arrInterfaceInfoValueWriteTo[byReadWriteArrayNumber].arrValue[uiLPWriteValueFromArray_WriteAds]),24) AND 16#FFFFFFFF);
								arrBufferWrite_WriteAds[arrCounterWriteValueInArray_WriteAds[3]] := UDINT_TO_BYTE(SHR(STRING_TO_UDINT(Lynus_Standards.GVL_Communicator.arrInterfaceInfoValueWriteTo[byReadWriteArrayNumber].arrValue[uiLPWriteValueFromArray_WriteAds]),16) AND 16#FFFFFFFF);
								arrBufferWrite_WriteAds[arrCounterWriteValueInArray_WriteAds[2]] := UDINT_TO_BYTE(SHR(STRING_TO_UDINT(Lynus_Standards.GVL_Communicator.arrInterfaceInfoValueWriteTo[byReadWriteArrayNumber].arrValue[uiLPWriteValueFromArray_WriteAds]),8) AND 16#FFFFFFFF);
								arrBufferWrite_WriteAds[arrCounterWriteValueInArray_WriteAds[1]] := UDINT_TO_BYTE(STRING_TO_UDINT(Lynus_Standards.GVL_Communicator.arrInterfaceInfoValueWriteTo[byReadWriteArrayNumber].arrValue[uiLPWriteValueFromArray_WriteAds]) AND 16#FFFFFFFF);  
						arrCounterWriteValueInArray_WriteAds[1] := arrCounterWriteValueInArray_WriteAds[1] + 4; arrCounterWriteValueInArray_WriteAds[2] := arrCounterWriteValueInArray_WriteAds[2] + 4;
							arrCounterWriteValueInArray_WriteAds[3] := arrCounterWriteValueInArray_WriteAds[3] + 4; arrCounterWriteValueInArray_WriteAds[4] := arrCounterWriteValueInArray_WriteAds[4] + 4;
								uiSizeToWrite_WriteAds := 4 * Lynus_Standards.GVL_Communicator.arrInterfaceInfoValueWriteTo[byReadWriteArrayNumber].uiSizeArray;	
									byCounterReceivedValueOK_WriteAds := byCounterReceivedValueOK_WriteAds + 1;
										byCounterReceivedValueOK_WriteAds := LIMIT(0,byCounterReceivedValueOK_WriteAds,Lynus_Standards.Constants_Communicator.bySizeOfValueArray);
											IF byCounterReceivedValueOK_WriteAds >= Lynus_Standards.GVL_Communicator.arrInterfaceInfoValueWriteTo[byReadWriteArrayNumber].uiSizeArray THEN bValueValid_WriteAds := TRUE; END_IF  
					END_IF
				END_FOR
			END_IF
			//Type LINT
			IF Lynus_Standards.GVL_Communicator.arrInterfaceInfoValueWriteTo[byReadWriteArrayNumber].uiSizeArray <= Lynus_Standards.Constants_Communicator.bySizeOfValueArray AND FIND(Lynus_Standards.GVL_Communicator.arrInterfaceInfoValueWriteTo[byReadWriteArrayNumber].sSymbolType,'OF LINT') <> 0 THEN
				FOR uiLPWriteValueFromArray_WriteAds := 1 TO Lynus_Standards.GVL_Communicator.arrInterfaceInfoValueWriteTo[byReadWriteArrayNumber].uiSizeArray BY 1 DO 
					IF TO_LINT(Lynus_Standards.GVL_Communicator.arrInterfaceInfoValueWriteTo[byReadWriteArrayNumber].arrValue[uiLPWriteValueFromArray_WriteAds]) >= -9223372036854775808 AND TO_LINT(Lynus_Standards.GVL_Communicator.arrInterfaceInfoValueWriteTo[byReadWriteArrayNumber].arrValue[uiLPWriteValueFromArray_WriteAds]) <= 9223372036854775807 THEN   
						arrCounterWriteValueInArray_WriteAds[1] := LIMIT(1,arrCounterWriteValueInArray_WriteAds[1],2000); arrCounterWriteValueInArray_WriteAds[2] := LIMIT(2,arrCounterWriteValueInArray_WriteAds[2],2000);
							arrCounterWriteValueInArray_WriteAds[3] := LIMIT(3,arrCounterWriteValueInArray_WriteAds[3],2000); arrCounterWriteValueInArray_WriteAds[4] := LIMIT(4,arrCounterWriteValueInArray_WriteAds[4],2000);	
								arrCounterWriteValueInArray_WriteAds[5] := LIMIT(5,arrCounterWriteValueInArray_WriteAds[5],2000); arrCounterWriteValueInArray_WriteAds[6] := LIMIT(6,arrCounterWriteValueInArray_WriteAds[6],2000);
									arrCounterWriteValueInArray_WriteAds[7] := LIMIT(7,arrCounterWriteValueInArray_WriteAds[7],2000); arrCounterWriteValueInArray_WriteAds[8] := LIMIT(8,arrCounterWriteValueInArray_WriteAds[8],2000);	
										arrBufferWrite_WriteAds[arrCounterWriteValueInArray_WriteAds[8]] := ULINT_TO_BYTE(SHR(LINT_TO_ULINT(STRING_TO_LINT(Lynus_Standards.GVL_Communicator.arrInterfaceInfoValueWriteTo[byReadWriteArrayNumber].arrValue[uiLPWriteValueFromArray_WriteAds])),56) AND 16#FFFFFFFFFFFFFFFF);
										arrBufferWrite_WriteAds[arrCounterWriteValueInArray_WriteAds[7]] := ULINT_TO_BYTE(SHR(LINT_TO_ULINT(STRING_TO_LINT(Lynus_Standards.GVL_Communicator.arrInterfaceInfoValueWriteTo[byReadWriteArrayNumber].arrValue[uiLPWriteValueFromArray_WriteAds])),48) AND 16#FFFFFFFFFFFFFFFF);
										arrBufferWrite_WriteAds[arrCounterWriteValueInArray_WriteAds[6]] := ULINT_TO_BYTE(SHR(LINT_TO_ULINT(STRING_TO_LINT(Lynus_Standards.GVL_Communicator.arrInterfaceInfoValueWriteTo[byReadWriteArrayNumber].arrValue[uiLPWriteValueFromArray_WriteAds])),40) AND 16#FFFFFFFFFFFFFFFF);
										arrBufferWrite_WriteAds[arrCounterWriteValueInArray_WriteAds[5]] := ULINT_TO_BYTE(SHR(LINT_TO_ULINT(STRING_TO_LINT(Lynus_Standards.GVL_Communicator.arrInterfaceInfoValueWriteTo[byReadWriteArrayNumber].arrValue[uiLPWriteValueFromArray_WriteAds])),32) AND 16#FFFFFFFFFFFFFFFF);
										arrBufferWrite_WriteAds[arrCounterWriteValueInArray_WriteAds[4]] := ULINT_TO_BYTE(SHR(LINT_TO_ULINT(STRING_TO_LINT(Lynus_Standards.GVL_Communicator.arrInterfaceInfoValueWriteTo[byReadWriteArrayNumber].arrValue[uiLPWriteValueFromArray_WriteAds])),24) AND 16#FFFFFFFFFFFFFFFF);
										arrBufferWrite_WriteAds[arrCounterWriteValueInArray_WriteAds[3]] := ULINT_TO_BYTE(SHR(LINT_TO_ULINT(STRING_TO_LINT(Lynus_Standards.GVL_Communicator.arrInterfaceInfoValueWriteTo[byReadWriteArrayNumber].arrValue[uiLPWriteValueFromArray_WriteAds])),16) AND 16#FFFFFFFFFFFFFFFF);
										arrBufferWrite_WriteAds[arrCounterWriteValueInArray_WriteAds[2]] := ULINT_TO_BYTE(SHR(LINT_TO_ULINT(STRING_TO_LINT(Lynus_Standards.GVL_Communicator.arrInterfaceInfoValueWriteTo[byReadWriteArrayNumber].arrValue[uiLPWriteValueFromArray_WriteAds])),8) AND 16#FFFFFFFFFFFFFFFF);
										arrBufferWrite_WriteAds[arrCounterWriteValueInArray_WriteAds[1]] := ULINT_TO_BYTE(LINT_TO_ULINT(STRING_TO_LINT(Lynus_Standards.GVL_Communicator.arrInterfaceInfoValueWriteTo[byReadWriteArrayNumber].arrValue[uiLPWriteValueFromArray_WriteAds])) AND 16#FFFFFFFFFFFFFFFF);
						arrCounterWriteValueInArray_WriteAds[1] := arrCounterWriteValueInArray_WriteAds[1] + 8; arrCounterWriteValueInArray_WriteAds[2] := arrCounterWriteValueInArray_WriteAds[2] + 8;
							arrCounterWriteValueInArray_WriteAds[3] := arrCounterWriteValueInArray_WriteAds[3] + 8; arrCounterWriteValueInArray_WriteAds[4] := arrCounterWriteValueInArray_WriteAds[4] + 8;
								arrCounterWriteValueInArray_WriteAds[5] := arrCounterWriteValueInArray_WriteAds[5] + 8; arrCounterWriteValueInArray_WriteAds[6] := arrCounterWriteValueInArray_WriteAds[6] + 8;
									arrCounterWriteValueInArray_WriteAds[7] := arrCounterWriteValueInArray_WriteAds[7] + 8; arrCounterWriteValueInArray_WriteAds[8] := arrCounterWriteValueInArray_WriteAds[8] + 8;
										uiSizeToWrite_WriteAds := 8 * Lynus_Standards.GVL_Communicator.arrInterfaceInfoValueWriteTo[byReadWriteArrayNumber].uiSizeArray;	
											byCounterReceivedValueOK_WriteAds := byCounterReceivedValueOK_WriteAds + 1;
												byCounterReceivedValueOK_WriteAds := LIMIT(0,byCounterReceivedValueOK_WriteAds,Lynus_Standards.Constants_Communicator.bySizeOfValueArray);
													IF byCounterReceivedValueOK_WriteAds >= Lynus_Standards.GVL_Communicator.arrInterfaceInfoValueWriteTo[byReadWriteArrayNumber].uiSizeArray THEN bValueValid_WriteAds := TRUE; END_IF  
					END_IF
				END_FOR
			END_IF
			//Type ULINT
			IF Lynus_Standards.GVL_Communicator.arrInterfaceInfoValueWriteTo[byReadWriteArrayNumber].uiSizeArray <= Lynus_Standards.Constants_Communicator.bySizeOfValueArray AND FIND(Lynus_Standards.GVL_Communicator.arrInterfaceInfoValueWriteTo[byReadWriteArrayNumber].sSymbolType,'OF ULINT') <> 0 THEN
				FOR uiLPWriteValueFromArray_WriteAds := 1 TO Lynus_Standards.GVL_Communicator.arrInterfaceInfoValueWriteTo[byReadWriteArrayNumber].uiSizeArray BY 1 DO 
					IF TO_ULINT(Lynus_Standards.GVL_Communicator.arrInterfaceInfoValueWriteTo[byReadWriteArrayNumber].arrValue[uiLPWriteValueFromArray_WriteAds]) >= 0 AND TO_ULINT(Lynus_Standards.GVL_Communicator.arrInterfaceInfoValueWriteTo[byReadWriteArrayNumber].arrValue[uiLPWriteValueFromArray_WriteAds]) <= 18446744073709551615 THEN   
						arrCounterWriteValueInArray_WriteAds[1] := LIMIT(1,arrCounterWriteValueInArray_WriteAds[1],2000); arrCounterWriteValueInArray_WriteAds[2] := LIMIT(2,arrCounterWriteValueInArray_WriteAds[2],2000);
							arrCounterWriteValueInArray_WriteAds[3] := LIMIT(3,arrCounterWriteValueInArray_WriteAds[3],2000); arrCounterWriteValueInArray_WriteAds[4] := LIMIT(4,arrCounterWriteValueInArray_WriteAds[4],2000);	
								arrCounterWriteValueInArray_WriteAds[5] := LIMIT(5,arrCounterWriteValueInArray_WriteAds[5],2000); arrCounterWriteValueInArray_WriteAds[6] := LIMIT(6,arrCounterWriteValueInArray_WriteAds[6],2000);
									arrCounterWriteValueInArray_WriteAds[7] := LIMIT(7,arrCounterWriteValueInArray_WriteAds[7],2000); arrCounterWriteValueInArray_WriteAds[8] := LIMIT(8,arrCounterWriteValueInArray_WriteAds[8],2000);	
										arrBufferWrite_WriteAds[arrCounterWriteValueInArray_WriteAds[8]] := ULINT_TO_BYTE(SHR(STRING_TO_ULINT(Lynus_Standards.GVL_Communicator.arrInterfaceInfoValueWriteTo[byReadWriteArrayNumber].arrValue[uiLPWriteValueFromArray_WriteAds]),56) AND 16#FFFFFFFFFFFFFFFF);
										arrBufferWrite_WriteAds[arrCounterWriteValueInArray_WriteAds[7]] := ULINT_TO_BYTE(SHR(STRING_TO_ULINT(Lynus_Standards.GVL_Communicator.arrInterfaceInfoValueWriteTo[byReadWriteArrayNumber].arrValue[uiLPWriteValueFromArray_WriteAds]),48) AND 16#FFFFFFFFFFFFFFFF);
										arrBufferWrite_WriteAds[arrCounterWriteValueInArray_WriteAds[6]] := ULINT_TO_BYTE(SHR(STRING_TO_ULINT(Lynus_Standards.GVL_Communicator.arrInterfaceInfoValueWriteTo[byReadWriteArrayNumber].arrValue[uiLPWriteValueFromArray_WriteAds]),40) AND 16#FFFFFFFFFFFFFFFF);
										arrBufferWrite_WriteAds[arrCounterWriteValueInArray_WriteAds[5]] := ULINT_TO_BYTE(SHR(STRING_TO_ULINT(Lynus_Standards.GVL_Communicator.arrInterfaceInfoValueWriteTo[byReadWriteArrayNumber].arrValue[uiLPWriteValueFromArray_WriteAds]),32) AND 16#FFFFFFFFFFFFFFFF);
										arrBufferWrite_WriteAds[arrCounterWriteValueInArray_WriteAds[4]] := ULINT_TO_BYTE(SHR(STRING_TO_ULINT(Lynus_Standards.GVL_Communicator.arrInterfaceInfoValueWriteTo[byReadWriteArrayNumber].arrValue[uiLPWriteValueFromArray_WriteAds]),24) AND 16#FFFFFFFFFFFFFFFF);
										arrBufferWrite_WriteAds[arrCounterWriteValueInArray_WriteAds[3]] := ULINT_TO_BYTE(SHR(STRING_TO_ULINT(Lynus_Standards.GVL_Communicator.arrInterfaceInfoValueWriteTo[byReadWriteArrayNumber].arrValue[uiLPWriteValueFromArray_WriteAds]),16) AND 16#FFFFFFFFFFFFFFFF);
										arrBufferWrite_WriteAds[arrCounterWriteValueInArray_WriteAds[2]] := ULINT_TO_BYTE(SHR(STRING_TO_ULINT(Lynus_Standards.GVL_Communicator.arrInterfaceInfoValueWriteTo[byReadWriteArrayNumber].arrValue[uiLPWriteValueFromArray_WriteAds]),8) AND 16#FFFFFFFFFFFFFFFF);
										arrBufferWrite_WriteAds[arrCounterWriteValueInArray_WriteAds[1]] := ULINT_TO_BYTE(STRING_TO_ULINT(Lynus_Standards.GVL_Communicator.arrInterfaceInfoValueWriteTo[byReadWriteArrayNumber].arrValue[uiLPWriteValueFromArray_WriteAds]) AND 16#FFFFFFFFFFFFFFFF);
						arrCounterWriteValueInArray_WriteAds[1] := arrCounterWriteValueInArray_WriteAds[1] + 8; arrCounterWriteValueInArray_WriteAds[2] := arrCounterWriteValueInArray_WriteAds[2] + 8;
							arrCounterWriteValueInArray_WriteAds[3] := arrCounterWriteValueInArray_WriteAds[3] + 8; arrCounterWriteValueInArray_WriteAds[4] := arrCounterWriteValueInArray_WriteAds[4] + 8;
								arrCounterWriteValueInArray_WriteAds[5] := arrCounterWriteValueInArray_WriteAds[5] + 8; arrCounterWriteValueInArray_WriteAds[6] := arrCounterWriteValueInArray_WriteAds[6] + 8;
									arrCounterWriteValueInArray_WriteAds[7] := arrCounterWriteValueInArray_WriteAds[7] + 8; arrCounterWriteValueInArray_WriteAds[8] := arrCounterWriteValueInArray_WriteAds[8] + 8;
										uiSizeToWrite_WriteAds := 8 * Lynus_Standards.GVL_Communicator.arrInterfaceInfoValueWriteTo[byReadWriteArrayNumber].uiSizeArray;	
											byCounterReceivedValueOK_WriteAds := byCounterReceivedValueOK_WriteAds + 1;
												byCounterReceivedValueOK_WriteAds := LIMIT(0,byCounterReceivedValueOK_WriteAds,Lynus_Standards.Constants_Communicator.bySizeOfValueArray);
													IF byCounterReceivedValueOK_WriteAds >= Lynus_Standards.GVL_Communicator.arrInterfaceInfoValueWriteTo[byReadWriteArrayNumber].uiSizeArray THEN bValueValid_WriteAds := TRUE; END_IF  
					END_IF
				END_FOR
			END_IF
			//Type LWORD
			IF Lynus_Standards.GVL_Communicator.arrInterfaceInfoValueWriteTo[byReadWriteArrayNumber].uiSizeArray <= Lynus_Standards.Constants_Communicator.bySizeOfValueArray AND FIND(Lynus_Standards.GVL_Communicator.arrInterfaceInfoValueWriteTo[byReadWriteArrayNumber].sSymbolType,'OF LWORD') <> 0 THEN
				FOR uiLPWriteValueFromArray_WriteAds := 1 TO Lynus_Standards.GVL_Communicator.arrInterfaceInfoValueWriteTo[byReadWriteArrayNumber].uiSizeArray BY 1 DO 
					IF TO_ULINT(Lynus_Standards.GVL_Communicator.arrInterfaceInfoValueWriteTo[byReadWriteArrayNumber].arrValue[uiLPWriteValueFromArray_WriteAds]) >= 0 AND TO_ULINT(Lynus_Standards.GVL_Communicator.arrInterfaceInfoValueWriteTo[byReadWriteArrayNumber].arrValue[uiLPWriteValueFromArray_WriteAds]) <= 18446744073709551615 THEN   
						arrCounterWriteValueInArray_WriteAds[1] := LIMIT(1,arrCounterWriteValueInArray_WriteAds[1],2000); arrCounterWriteValueInArray_WriteAds[2] := LIMIT(2,arrCounterWriteValueInArray_WriteAds[2],2000);
							arrCounterWriteValueInArray_WriteAds[3] := LIMIT(3,arrCounterWriteValueInArray_WriteAds[3],2000); arrCounterWriteValueInArray_WriteAds[4] := LIMIT(4,arrCounterWriteValueInArray_WriteAds[4],2000);	
								arrCounterWriteValueInArray_WriteAds[5] := LIMIT(5,arrCounterWriteValueInArray_WriteAds[5],2000); arrCounterWriteValueInArray_WriteAds[6] := LIMIT(6,arrCounterWriteValueInArray_WriteAds[6],2000);
									arrCounterWriteValueInArray_WriteAds[7] := LIMIT(7,arrCounterWriteValueInArray_WriteAds[7],2000); arrCounterWriteValueInArray_WriteAds[8] := LIMIT(8,arrCounterWriteValueInArray_WriteAds[8],2000);	
										arrBufferWrite_WriteAds[arrCounterWriteValueInArray_WriteAds[8]] := ULINT_TO_BYTE(SHR(STRING_TO_ULINT(Lynus_Standards.GVL_Communicator.arrInterfaceInfoValueWriteTo[byReadWriteArrayNumber].arrValue[uiLPWriteValueFromArray_WriteAds]),56) AND 16#FFFFFFFFFFFFFFFF);
										arrBufferWrite_WriteAds[arrCounterWriteValueInArray_WriteAds[7]] := ULINT_TO_BYTE(SHR(STRING_TO_ULINT(Lynus_Standards.GVL_Communicator.arrInterfaceInfoValueWriteTo[byReadWriteArrayNumber].arrValue[uiLPWriteValueFromArray_WriteAds]),48) AND 16#FFFFFFFFFFFFFFFF);
										arrBufferWrite_WriteAds[arrCounterWriteValueInArray_WriteAds[6]] := ULINT_TO_BYTE(SHR(STRING_TO_ULINT(Lynus_Standards.GVL_Communicator.arrInterfaceInfoValueWriteTo[byReadWriteArrayNumber].arrValue[uiLPWriteValueFromArray_WriteAds]),40) AND 16#FFFFFFFFFFFFFFFF);
										arrBufferWrite_WriteAds[arrCounterWriteValueInArray_WriteAds[5]] := ULINT_TO_BYTE(SHR(STRING_TO_ULINT(Lynus_Standards.GVL_Communicator.arrInterfaceInfoValueWriteTo[byReadWriteArrayNumber].arrValue[uiLPWriteValueFromArray_WriteAds]),32) AND 16#FFFFFFFFFFFFFFFF);
										arrBufferWrite_WriteAds[arrCounterWriteValueInArray_WriteAds[4]] := ULINT_TO_BYTE(SHR(STRING_TO_ULINT(Lynus_Standards.GVL_Communicator.arrInterfaceInfoValueWriteTo[byReadWriteArrayNumber].arrValue[uiLPWriteValueFromArray_WriteAds]),24) AND 16#FFFFFFFFFFFFFFFF);
										arrBufferWrite_WriteAds[arrCounterWriteValueInArray_WriteAds[3]] := ULINT_TO_BYTE(SHR(STRING_TO_ULINT(Lynus_Standards.GVL_Communicator.arrInterfaceInfoValueWriteTo[byReadWriteArrayNumber].arrValue[uiLPWriteValueFromArray_WriteAds]),16) AND 16#FFFFFFFFFFFFFFFF);
										arrBufferWrite_WriteAds[arrCounterWriteValueInArray_WriteAds[2]] := ULINT_TO_BYTE(SHR(STRING_TO_ULINT(Lynus_Standards.GVL_Communicator.arrInterfaceInfoValueWriteTo[byReadWriteArrayNumber].arrValue[uiLPWriteValueFromArray_WriteAds]),8) AND 16#FFFFFFFFFFFFFFFF);
										arrBufferWrite_WriteAds[arrCounterWriteValueInArray_WriteAds[1]] := ULINT_TO_BYTE(STRING_TO_ULINT(Lynus_Standards.GVL_Communicator.arrInterfaceInfoValueWriteTo[byReadWriteArrayNumber].arrValue[uiLPWriteValueFromArray_WriteAds]) AND 16#FFFFFFFFFFFFFFFF);
						arrCounterWriteValueInArray_WriteAds[1] := arrCounterWriteValueInArray_WriteAds[1] + 8; arrCounterWriteValueInArray_WriteAds[2] := arrCounterWriteValueInArray_WriteAds[2] + 8;
							arrCounterWriteValueInArray_WriteAds[3] := arrCounterWriteValueInArray_WriteAds[3] + 8; arrCounterWriteValueInArray_WriteAds[4] := arrCounterWriteValueInArray_WriteAds[4] + 8;
								arrCounterWriteValueInArray_WriteAds[5] := arrCounterWriteValueInArray_WriteAds[5] + 8; arrCounterWriteValueInArray_WriteAds[6] := arrCounterWriteValueInArray_WriteAds[6] + 8;
									arrCounterWriteValueInArray_WriteAds[7] := arrCounterWriteValueInArray_WriteAds[7] + 8; arrCounterWriteValueInArray_WriteAds[8] := arrCounterWriteValueInArray_WriteAds[8] + 8;
										uiSizeToWrite_WriteAds := 8 * Lynus_Standards.GVL_Communicator.arrInterfaceInfoValueWriteTo[byReadWriteArrayNumber].uiSizeArray;	
											byCounterReceivedValueOK_WriteAds := byCounterReceivedValueOK_WriteAds + 1;
												byCounterReceivedValueOK_WriteAds := LIMIT(0,byCounterReceivedValueOK_WriteAds,Lynus_Standards.Constants_Communicator.bySizeOfValueArray);
													IF byCounterReceivedValueOK_WriteAds >= Lynus_Standards.GVL_Communicator.arrInterfaceInfoValueWriteTo[byReadWriteArrayNumber].uiSizeArray THEN bValueValid_WriteAds := TRUE; END_IF  
					END_IF
				END_FOR
			END_IF
			//Type REAL
			IF Lynus_Standards.GVL_Communicator.arrInterfaceInfoValueWriteTo[byReadWriteArrayNumber].uiSizeArray <= Lynus_Standards.Constants_Communicator.bySizeOfValueArray AND FIND(Lynus_Standards.GVL_Communicator.arrInterfaceInfoValueWriteTo[byReadWriteArrayNumber].sSymbolType,'OF REAL') <> 0 THEN
				FOR uiLPWriteValueFromArray_WriteAds := 1 TO Lynus_Standards.GVL_Communicator.arrInterfaceInfoValueWriteTo[byReadWriteArrayNumber].uiSizeArray BY 1 DO 
					IF LEN(Lynus_Standards.GVL_Communicator.arrInterfaceInfoValueWriteTo[byReadWriteArrayNumber].arrValue[uiLPWriteValueFromArray_WriteAds]) <= 30 AND TO_LREAL(Lynus_Standards.GVL_Communicator.arrInterfaceInfoValueWriteTo[byReadWriteArrayNumber].arrValue[uiLPWriteValueFromArray_WriteAds]) >= -3.40282326E+38 AND TO_LREAL(Lynus_Standards.GVL_Communicator.arrInterfaceInfoValueWriteTo[byReadWriteArrayNumber].arrValue[uiLPWriteValueFromArray_WriteAds]) <= 3.40282326E+38 THEN   
						rRealValueCheckBeforWrite_WriteAds := STRING_TO_REAL(Lynus_Standards.GVL_Communicator.arrInterfaceInfoValueWriteTo[byReadWriteArrayNumber].arrValue[uiLPWriteValueFromArray_WriteAds]); 							
							IF IsFinite(F_REAL(rRealValueCheckBeforWrite_WriteAds)) THEN 
								unConvertDWORD_TO_REAL_WriteAds.rValueFloat := STRING_TO_REAL(Lynus_Standards.GVL_Communicator.arrInterfaceInfoValueWriteTo[byReadWriteArrayNumber].arrValue[uiLPWriteValueFromArray_WriteAds]);
									arrCounterWriteValueInArray_WriteAds[1] := LIMIT(1,arrCounterWriteValueInArray_WriteAds[1],2000); arrCounterWriteValueInArray_WriteAds[2] := LIMIT(2,arrCounterWriteValueInArray_WriteAds[2],2000);
										arrCounterWriteValueInArray_WriteAds[3] := LIMIT(3,arrCounterWriteValueInArray_WriteAds[3],2000); arrCounterWriteValueInArray_WriteAds[4] := LIMIT(4,arrCounterWriteValueInArray_WriteAds[4],2000);	
											arrBufferWrite_WriteAds[arrCounterWriteValueInArray_WriteAds[4]] := UDINT_TO_BYTE((SHR(DWORD_TO_UDINT(unConvertDWORD_TO_REAL_WriteAds.dwRawValue),24) AND 16#FFFFFFFF));
											arrBufferWrite_WriteAds[arrCounterWriteValueInArray_WriteAds[3]] := UDINT_TO_BYTE((SHR(DWORD_TO_UDINT(unConvertDWORD_TO_REAL_WriteAds.dwRawValue),16) AND 16#FFFFFFFF));
											arrBufferWrite_WriteAds[arrCounterWriteValueInArray_WriteAds[2]] := UDINT_TO_BYTE((SHR(DWORD_TO_UDINT(unConvertDWORD_TO_REAL_WriteAds.dwRawValue),8) AND 16#FFFFFFFF));
											arrBufferWrite_WriteAds[arrCounterWriteValueInArray_WriteAds[1]] := UDINT_TO_BYTE(DWORD_TO_UDINT(unConvertDWORD_TO_REAL_WriteAds.dwRawValue) AND 16#FFFFFFFF);  
												arrCounterWriteValueInArray_WriteAds[1] := arrCounterWriteValueInArray_WriteAds[1] + 4; arrCounterWriteValueInArray_WriteAds[2] := arrCounterWriteValueInArray_WriteAds[2] + 4;
													arrCounterWriteValueInArray_WriteAds[3] := arrCounterWriteValueInArray_WriteAds[3] + 4; arrCounterWriteValueInArray_WriteAds[4] := arrCounterWriteValueInArray_WriteAds[4] + 4;
														uiSizeToWrite_WriteAds := 4 * Lynus_Standards.GVL_Communicator.arrInterfaceInfoValueWriteTo[byReadWriteArrayNumber].uiSizeArray;	
															byCounterReceivedValueOK_WriteAds := byCounterReceivedValueOK_WriteAds + 1;
																byCounterReceivedValueOK_WriteAds := LIMIT(0,byCounterReceivedValueOK_WriteAds,Lynus_Standards.Constants_Communicator.bySizeOfValueArray);
																	IF byCounterReceivedValueOK_WriteAds >= Lynus_Standards.GVL_Communicator.arrInterfaceInfoValueWriteTo[byReadWriteArrayNumber].uiSizeArray THEN bValueValid_WriteAds := TRUE; END_IF  
							END_IF
					END_IF
				END_FOR
			END_IF
			//Type LREAL
			IF Lynus_Standards.GVL_Communicator.arrInterfaceInfoValueWriteTo[byReadWriteArrayNumber].uiSizeArray <= Lynus_Standards.Constants_Communicator.bySizeOfValueArray AND FIND(Lynus_Standards.GVL_Communicator.arrInterfaceInfoValueWriteTo[byReadWriteArrayNumber].sSymbolType,'OF LREAL') <> 0 THEN
				FOR uiLPWriteValueFromArray_WriteAds := 1 TO Lynus_Standards.GVL_Communicator.arrInterfaceInfoValueWriteTo[byReadWriteArrayNumber].uiSizeArray BY 1 DO 
					IF LEN(Lynus_Standards.GVL_Communicator.arrInterfaceInfoValueWriteTo[byReadWriteArrayNumber].arrValue[uiLPWriteValueFromArray_WriteAds]) <= 30 AND TO_LREAL(Lynus_Standards.GVL_Communicator.arrInterfaceInfoValueWriteTo[byReadWriteArrayNumber].arrValue[uiLPWriteValueFromArray_WriteAds]) >= -1.7976931348623157E+307 AND TO_LREAL(Lynus_Standards.GVL_Communicator.arrInterfaceInfoValueWriteTo[byReadWriteArrayNumber].arrValue[uiLPWriteValueFromArray_WriteAds]) <= 1.7976931348623157E+307 THEN   
						lrRealValueCheckBeforWrite_WriteAds := STRING_TO_LREAL(Lynus_Standards.GVL_Communicator.arrInterfaceInfoValueWriteTo[byReadWriteArrayNumber].arrValue[uiLPWriteValueFromArray_WriteAds]); 							
							IF IsFinite(F_LREAL(lrRealValueCheckBeforWrite_WriteAds)) THEN 
								unConvertULINT_TO_LREAL_WriteAds.lrValueFloat := STRING_TO_LREAL(Lynus_Standards.GVL_Communicator.arrInterfaceInfoValueWriteTo[byReadWriteArrayNumber].arrValue[uiLPWriteValueFromArray_WriteAds]);
									arrCounterWriteValueInArray_WriteAds[1] := LIMIT(1,arrCounterWriteValueInArray_WriteAds[1],2000); arrCounterWriteValueInArray_WriteAds[2] := LIMIT(2,arrCounterWriteValueInArray_WriteAds[2],2000);
										arrCounterWriteValueInArray_WriteAds[3] := LIMIT(3,arrCounterWriteValueInArray_WriteAds[3],2000); arrCounterWriteValueInArray_WriteAds[4] := LIMIT(4,arrCounterWriteValueInArray_WriteAds[4],2000);	
											arrCounterWriteValueInArray_WriteAds[5] := LIMIT(5,arrCounterWriteValueInArray_WriteAds[5],2000); arrCounterWriteValueInArray_WriteAds[6] := LIMIT(6,arrCounterWriteValueInArray_WriteAds[6],2000);
												arrCounterWriteValueInArray_WriteAds[7] := LIMIT(7,arrCounterWriteValueInArray_WriteAds[7],2000); arrCounterWriteValueInArray_WriteAds[8] := LIMIT(8,arrCounterWriteValueInArray_WriteAds[8],2000);	
													arrBufferWrite_WriteAds[arrCounterWriteValueInArray_WriteAds[8]] := LWORD_TO_BYTE((SHR(ULINT_TO_LWORD(unConvertULINT_TO_LREAL_WriteAds.uliRawValue),56) AND 16#FFFFFFFFFFFFFFFF));
													arrBufferWrite_WriteAds[arrCounterWriteValueInArray_WriteAds[7]] := LWORD_TO_BYTE((SHR(ULINT_TO_LWORD(unConvertULINT_TO_LREAL_WriteAds.uliRawValue),48) AND 16#FFFFFFFFFFFFFFFF));
													arrBufferWrite_WriteAds[arrCounterWriteValueInArray_WriteAds[6]] := LWORD_TO_BYTE((SHR(ULINT_TO_LWORD(unConvertULINT_TO_LREAL_WriteAds.uliRawValue),40) AND 16#FFFFFFFFFFFFFFFF));
													arrBufferWrite_WriteAds[arrCounterWriteValueInArray_WriteAds[5]] := LWORD_TO_BYTE((SHR(ULINT_TO_LWORD(unConvertULINT_TO_LREAL_WriteAds.uliRawValue),32) AND 16#FFFFFFFFFFFFFFFF));
													arrBufferWrite_WriteAds[arrCounterWriteValueInArray_WriteAds[4]] := LWORD_TO_BYTE((SHR(ULINT_TO_LWORD(unConvertULINT_TO_LREAL_WriteAds.uliRawValue),24) AND 16#FFFFFFFFFFFFFFFF));
													arrBufferWrite_WriteAds[arrCounterWriteValueInArray_WriteAds[3]] := LWORD_TO_BYTE((SHR(ULINT_TO_LWORD(unConvertULINT_TO_LREAL_WriteAds.uliRawValue),16) AND 16#FFFFFFFFFFFFFFFF));
													arrBufferWrite_WriteAds[arrCounterWriteValueInArray_WriteAds[2]] := LWORD_TO_BYTE((SHR(ULINT_TO_LWORD(unConvertULINT_TO_LREAL_WriteAds.uliRawValue),8) AND 16#FFFFFFFFFFFFFFFF));
													arrBufferWrite_WriteAds[arrCounterWriteValueInArray_WriteAds[1]] := LWORD_TO_BYTE(ULINT_TO_LWORD(unConvertULINT_TO_LREAL_WriteAds.uliRawValue) AND 16#FFFFFFFFFFFFFFFF);  
									arrCounterWriteValueInArray_WriteAds[1] := arrCounterWriteValueInArray_WriteAds[1] + 8; arrCounterWriteValueInArray_WriteAds[2] := arrCounterWriteValueInArray_WriteAds[2] + 8;
										arrCounterWriteValueInArray_WriteAds[3] := arrCounterWriteValueInArray_WriteAds[3] + 8; arrCounterWriteValueInArray_WriteAds[4] := arrCounterWriteValueInArray_WriteAds[4] + 8;
											arrCounterWriteValueInArray_WriteAds[5] := arrCounterWriteValueInArray_WriteAds[5] + 8; arrCounterWriteValueInArray_WriteAds[6] := arrCounterWriteValueInArray_WriteAds[6] + 8;
												arrCounterWriteValueInArray_WriteAds[7] := arrCounterWriteValueInArray_WriteAds[7] + 8; arrCounterWriteValueInArray_WriteAds[8] := arrCounterWriteValueInArray_WriteAds[8] + 8;
													uiSizeToWrite_WriteAds := 8 * Lynus_Standards.GVL_Communicator.arrInterfaceInfoValueWriteTo[byReadWriteArrayNumber].uiSizeArray;	
														byCounterReceivedValueOK_WriteAds := byCounterReceivedValueOK_WriteAds + 1;
															byCounterReceivedValueOK_WriteAds := LIMIT(0,byCounterReceivedValueOK_WriteAds,Lynus_Standards.Constants_Communicator.bySizeOfValueArray);
																IF byCounterReceivedValueOK_WriteAds >= Lynus_Standards.GVL_Communicator.arrInterfaceInfoValueWriteTo[byReadWriteArrayNumber].uiSizeArray THEN bValueValid_WriteAds := TRUE; END_IF  
							END_IF
					END_IF
				END_FOR
			END_IF
			//Type STRING(30)
			IF Lynus_Standards.GVL_Communicator.arrInterfaceInfoValueWriteTo[byReadWriteArrayNumber].uiSizeArray <= Lynus_Standards.Constants_Communicator.bySizeOfValueArray AND FIND(Lynus_Standards.GVL_Communicator.arrInterfaceInfoValueWriteTo[byReadWriteArrayNumber].sSymbolType,'OF STRING(30)') <> 0 THEN
				FOR uiLPWriteValueFromArray_WriteAds := 1 TO Lynus_Standards.GVL_Communicator.arrInterfaceInfoValueWriteTo[byReadWriteArrayNumber].uiSizeArray BY 1 DO   
					IF LEN(Lynus_Standards.GVL_Communicator.arrInterfaceInfoValueWriteTo[byReadWriteArrayNumber].arrValue[uiLPWriteValueFromArray_WriteAds]) <= 30 AND FIND(Lynus_Standards.GVL_Communicator.arrInterfaceInfoValueWriteTo[byReadWriteArrayNumber].arrValue[uiLPWriteValueFromArray_WriteAds],'#EMPTY#') = 0 THEN
						FOR byLPEncodeReceivedString_WriteAds := 1 TO 30 BY 1 DO 
							 uiCounterEncodeString_WriteAds := uiCounterEncodeString_WriteAds + 1;
								byCounterEncodeString_WriteAds := byCounterEncodeString_WriteAds + 1;
									byCounterEncodeString_WriteAds := LIMIT(1,byCounterEncodeString_WriteAds,30);
										uiCounterEncodeString_WriteAds := LIMIT(1,uiCounterEncodeString_WriteAds,2000);
											arrBufferWrite_WriteAds[uiCounterEncodeString_WriteAds] := F_ToASC(MID(Lynus_Standards.GVL_Communicator.arrInterfaceInfoValueWriteTo[byReadWriteArrayNumber].arrValue[uiLPWriteValueFromArray_WriteAds],1,byCounterEncodeString_WriteAds));
						END_FOR
					END_IF
					IF LEN(Lynus_Standards.GVL_Communicator.arrInterfaceInfoValueWriteTo[byReadWriteArrayNumber].arrValue[uiLPWriteValueFromArray_WriteAds]) <= 30 AND FIND(Lynus_Standards.GVL_Communicator.arrInterfaceInfoValueWriteTo[byReadWriteArrayNumber].arrValue[uiLPWriteValueFromArray_WriteAds],'#EMPTY#') <> 0 THEN
						FOR byLPEncodeReceivedString_WriteAds := 1 TO 30 BY 1 DO 
							 uiCounterEncodeString_WriteAds := uiCounterEncodeString_WriteAds + 1;
								byCounterEncodeString_WriteAds := byCounterEncodeString_WriteAds + 1;
									byCounterEncodeString_WriteAds := LIMIT(1,byCounterEncodeString_WriteAds,30);
										uiCounterEncodeString_WriteAds := LIMIT(1,uiCounterEncodeString_WriteAds,2000);
											arrBufferWrite_WriteAds[uiCounterEncodeString_WriteAds] := F_ToASC('');
						END_FOR	 
					END_IF
						byCounterEncodeString_WriteAds := 0;
							uiCounterEncodeString_WriteAds := uiCounterEncodeString_WriteAds + 1;
								uiSizeToWrite_WriteAds := 1 * uiCounterEncodeString_WriteAds;
									byCounterReceivedValueOK_WriteAds := byCounterReceivedValueOK_WriteAds + 1;
										byCounterReceivedValueOK_WriteAds := LIMIT(0,byCounterReceivedValueOK_WriteAds,Lynus_Standards.Constants_Communicator.bySizeOfValueArray);
											IF byCounterReceivedValueOK_WriteAds >= Lynus_Standards.GVL_Communicator.arrInterfaceInfoValueWriteTo[byReadWriteArrayNumber].uiSizeArray THEN bValueValid_WriteAds := TRUE; END_IF 	
				END_FOR
			END_IF
			//Type TIME and TIME_OF_DAY
			IF (Lynus_Standards.GVL_Communicator.arrInterfaceInfoValueWriteTo[byReadWriteArrayNumber].uiSizeArray <= Lynus_Standards.Constants_Communicator.bySizeOfValueArray AND (FIND(Lynus_Standards.GVL_Communicator.arrInterfaceInfoValueWriteTo[byReadWriteArrayNumber].sSymbolType,'OF TIME') <> 0 OR FIND(Lynus_Standards.GVL_Communicator.arrInterfaceInfoValueWriteTo[byReadWriteArrayNumber].sSymbolType,'OF TIME_OF_DAY') <> 0)) THEN
				FOR uiLPWriteValueFromArray_WriteAds := 1 TO Lynus_Standards.GVL_Communicator.arrInterfaceInfoValueWriteTo[byReadWriteArrayNumber].uiSizeArray BY 1 DO 
					IF TO_LWORD(Lynus_Standards.GVL_Communicator.arrInterfaceInfoValueWriteTo[byReadWriteArrayNumber].arrValue[uiLPWriteValueFromArray_WriteAds]) >= 0 AND TO_LWORD(Lynus_Standards.GVL_Communicator.arrInterfaceInfoValueWriteTo[byReadWriteArrayNumber].arrValue[uiLPWriteValueFromArray_WriteAds]) <= 4294967295 THEN   
						arrCounterWriteValueInArray_WriteAds[1] := LIMIT(1,arrCounterWriteValueInArray_WriteAds[1],2000); arrCounterWriteValueInArray_WriteAds[2] := LIMIT(2,arrCounterWriteValueInArray_WriteAds[2],2000);
							arrCounterWriteValueInArray_WriteAds[3] := LIMIT(3,arrCounterWriteValueInArray_WriteAds[3],2000); arrCounterWriteValueInArray_WriteAds[4] := LIMIT(4,arrCounterWriteValueInArray_WriteAds[4],2000);	
								arrBufferWrite_WriteAds[arrCounterWriteValueInArray_WriteAds[4]] := UDINT_TO_BYTE(SHR(STRING_TO_UDINT(Lynus_Standards.GVL_Communicator.arrInterfaceInfoValueWriteTo[byReadWriteArrayNumber].arrValue[uiLPWriteValueFromArray_WriteAds]),24) AND 16#FFFFFFFF);
								arrBufferWrite_WriteAds[arrCounterWriteValueInArray_WriteAds[3]] := UDINT_TO_BYTE(SHR(STRING_TO_UDINT(Lynus_Standards.GVL_Communicator.arrInterfaceInfoValueWriteTo[byReadWriteArrayNumber].arrValue[uiLPWriteValueFromArray_WriteAds]),16) AND 16#FFFFFFFF);
								arrBufferWrite_WriteAds[arrCounterWriteValueInArray_WriteAds[2]] := UDINT_TO_BYTE(SHR(STRING_TO_UDINT(Lynus_Standards.GVL_Communicator.arrInterfaceInfoValueWriteTo[byReadWriteArrayNumber].arrValue[uiLPWriteValueFromArray_WriteAds]),8) AND 16#FFFFFFFF);
								arrBufferWrite_WriteAds[arrCounterWriteValueInArray_WriteAds[1]] := UDINT_TO_BYTE(STRING_TO_UDINT(Lynus_Standards.GVL_Communicator.arrInterfaceInfoValueWriteTo[byReadWriteArrayNumber].arrValue[uiLPWriteValueFromArray_WriteAds]) AND 16#FFFFFFFF);  
						arrCounterWriteValueInArray_WriteAds[1] := arrCounterWriteValueInArray_WriteAds[1] + 4; arrCounterWriteValueInArray_WriteAds[2] := arrCounterWriteValueInArray_WriteAds[2] + 4;
							arrCounterWriteValueInArray_WriteAds[3] := arrCounterWriteValueInArray_WriteAds[3] + 4; arrCounterWriteValueInArray_WriteAds[4] := arrCounterWriteValueInArray_WriteAds[4] + 4;
								uiSizeToWrite_WriteAds := 4 * Lynus_Standards.GVL_Communicator.arrInterfaceInfoValueWriteTo[byReadWriteArrayNumber].uiSizeArray;	
									byCounterReceivedValueOK_WriteAds := byCounterReceivedValueOK_WriteAds + 1;
										byCounterReceivedValueOK_WriteAds := LIMIT(0,byCounterReceivedValueOK_WriteAds,Lynus_Standards.Constants_Communicator.bySizeOfValueArray);
											IF byCounterReceivedValueOK_WriteAds >= Lynus_Standards.GVL_Communicator.arrInterfaceInfoValueWriteTo[byReadWriteArrayNumber].uiSizeArray THEN bValueValid_WriteAds := TRUE; END_IF  
					END_IF
				END_FOR
			END_IF
			//Type DATE and DATE_AND_TIME
			IF (Lynus_Standards.GVL_Communicator.arrInterfaceInfoValueWriteTo[byReadWriteArrayNumber].uiSizeArray <= Lynus_Standards.Constants_Communicator.bySizeOfValueArray AND (FIND(Lynus_Standards.GVL_Communicator.arrInterfaceInfoValueWriteTo[byReadWriteArrayNumber].sSymbolType,'OF DATE') <> 0 OR FIND(Lynus_Standards.GVL_Communicator.arrInterfaceInfoValueWriteTo[byReadWriteArrayNumber].sSymbolType,'OF DATE_AND_TIME') <> 0)) THEN
				FOR uiLPWriteValueFromArray_WriteAds := 1 TO Lynus_Standards.GVL_Communicator.arrInterfaceInfoValueWriteTo[byReadWriteArrayNumber].uiSizeArray BY 1 DO 
					IF TO_LWORD(Lynus_Standards.GVL_Communicator.arrInterfaceInfoValueWriteTo[byReadWriteArrayNumber].arrValue[uiLPWriteValueFromArray_WriteAds]) >= 0 AND TO_LWORD(Lynus_Standards.GVL_Communicator.arrInterfaceInfoValueWriteTo[byReadWriteArrayNumber].arrValue[uiLPWriteValueFromArray_WriteAds]) <= 4294967295000 THEN 
						uliDate_WriteAds := STRING_TO_ULINT(Lynus_Standards.GVL_Communicator.arrInterfaceInfoValueWriteTo[byReadWriteArrayNumber].arrValue[uiLPWriteValueFromArray_WriteAds]);  
							udiDate_WriteAds := ULINT_TO_UDINT(uliDate_WriteAds / 1000);
								arrCounterWriteValueInArray_WriteAds[1] := LIMIT(1,arrCounterWriteValueInArray_WriteAds[1],2000); arrCounterWriteValueInArray_WriteAds[2] := LIMIT(2,arrCounterWriteValueInArray_WriteAds[2],2000);
									arrCounterWriteValueInArray_WriteAds[3] := LIMIT(3,arrCounterWriteValueInArray_WriteAds[3],2000); arrCounterWriteValueInArray_WriteAds[4] := LIMIT(4,arrCounterWriteValueInArray_WriteAds[4],2000);	
										arrBufferWrite_WriteAds[arrCounterWriteValueInArray_WriteAds[4]] := UDINT_TO_BYTE(SHR(udiDate_WriteAds,24) AND 16#FFFFFFFF);
										arrBufferWrite_WriteAds[arrCounterWriteValueInArray_WriteAds[3]] := UDINT_TO_BYTE(SHR(udiDate_WriteAds,16) AND 16#FFFFFFFF);
										arrBufferWrite_WriteAds[arrCounterWriteValueInArray_WriteAds[2]] := UDINT_TO_BYTE(SHR(udiDate_WriteAds,8) AND 16#FFFFFFFF);
										arrBufferWrite_WriteAds[arrCounterWriteValueInArray_WriteAds[1]] := UDINT_TO_BYTE(udiDate_WriteAds AND 16#FFFFFFFF);  
								arrCounterWriteValueInArray_WriteAds[1] := arrCounterWriteValueInArray_WriteAds[1] + 4; arrCounterWriteValueInArray_WriteAds[2] := arrCounterWriteValueInArray_WriteAds[2] + 4;
									arrCounterWriteValueInArray_WriteAds[3] := arrCounterWriteValueInArray_WriteAds[3] + 4; arrCounterWriteValueInArray_WriteAds[4] := arrCounterWriteValueInArray_WriteAds[4] + 4;
										uiSizeToWrite_WriteAds := 4 * Lynus_Standards.GVL_Communicator.arrInterfaceInfoValueWriteTo[byReadWriteArrayNumber].uiSizeArray;	
											byCounterReceivedValueOK_WriteAds := byCounterReceivedValueOK_WriteAds + 1;
												byCounterReceivedValueOK_WriteAds := LIMIT(0,byCounterReceivedValueOK_WriteAds,Lynus_Standards.Constants_Communicator.bySizeOfValueArray);
													IF byCounterReceivedValueOK_WriteAds >= Lynus_Standards.GVL_Communicator.arrInterfaceInfoValueWriteTo[byReadWriteArrayNumber].uiSizeArray THEN bValueValid_WriteAds := TRUE; END_IF  
					END_IF
				END_FOR
			END_IF
			
			IF timTimout_WriteAds.Q OR NOT bValueValid_WriteAds THEN 
				iState_WriteAds := 200; 
					IF NOT bValueValid_WriteAds THEN uiInternError_WriteAds := 1; END_IF 
			ELSE
				iState_WriteAds := 3;
					bValueValid_WriteAds := FALSE;
						byCounterEncodeString_WriteAds := 0; udiDate_WriteAds := 0; byCounterReceivedValueOK_WriteAds := 0; uiCounterEncodeString_WriteAds := 0; uliDate_WriteAds := 0;
							arrCounterWriteValueInArray_WriteAds[1] := 0; arrCounterWriteValueInArray_WriteAds[2] := 0; arrCounterWriteValueInArray_WriteAds[3] := 0; arrCounterWriteValueInArray_WriteAds[4] := 0;
								arrCounterWriteValueInArray_WriteAds[5] := 0; arrCounterWriteValueInArray_WriteAds[6] := 0; arrCounterWriteValueInArray_WriteAds[7] := 0; arrCounterWriteValueInArray_WriteAds[8] := 0;	
			END_IF
		
	3://Write Value
		IF Lynus_Standards.GVL_Communicator.arrCounterVariableInArray[byReadWriteArrayNumber] >= 1 AND Lynus_Standards.GVL_Communicator.arrCounterVariableInArray[byReadWriteArrayNumber] <= Lynus_Standards.Constants_Communicator.udiArraySizeMarkedSymobls THEN 
			FOR udiLPWriteInReadArrayForCheck_WriteADS := 1 TO Lynus_Standards.GVL_Communicator.arrCounterVariableInArray[byReadWriteArrayNumber] BY 1 DO 
				IF Lynus_Standards.GVL_Communicator.arrInterfaceInfoValueWriteTo[byReadWriteArrayNumber].sFullSymbolName = stADSRead_ReadAds[udiLPWriteInReadArrayForCheck_WriteADS].sFullSymbolName THEN
					stADSRead_ReadAds[udiLPWriteInReadArrayForCheck_WriteADS].arrValue := Lynus_Standards.GVL_Communicator.arrInterfaceInfoValueWriteTo[byReadWriteArrayNumber].arrValue; 
						stADSReadNew_ReadAds[udiLPWriteInReadArrayForCheck_WriteADS].arrValue := Lynus_Standards.GVL_Communicator.arrInterfaceInfoValueWriteTo[byReadWriteArrayNumber].arrValue;	
							EXIT;		
				END_IF
			END_FOR	
		END_IF
		
		//Extensions of the waiting step until data has been successfully written via ads so that the old value is not read back too quickly
		uiWaitBySymbolString_WriteAds := REAL_TO_UINT(F_Scalvalue(x:= UDINT_TO_REAL(udiCycleTime), x1:= 1, y1:= 25, x2:= 10, y2:= 1));
			uiWaitBySymbolString_WriteAds := LIMIT(1,uiWaitBySymbolString_WriteAds,25);
		
		IF Lynus_Standards.GVL_Communicator.arrInterfaceInfoValueWriteTo[byReadWriteArrayNumber].uiSizeArray > 2 THEN 
			uiWaitBySymbolString_WriteAds := uiWaitBySymbolString_WriteAds + Lynus_Standards.GVL_Communicator.arrInterfaceInfoValueWriteTo[byReadWriteArrayNumber].uiSizeArray * 8;
		ELSE
			uiWaitBySymbolString_WriteAds := uiWaitBySymbolString_WriteAds + 20;
		END_IF
	
		IF FIND(Lynus_Standards.GVL_Communicator.arrInterfaceInfoValueWriteTo[byReadWriteArrayNumber].sSymbolType,'OF STRING(30)') <> 0 THEN uiWaitBySymbolString_WriteAds := uiWaitBySymbolString_WriteAds + (Lynus_Standards.GVL_Communicator.arrInterfaceInfoValueWriteTo[byReadWriteArrayNumber].uiSizeArray * 8); END_IF
		
			uiWaitBySymbolString_WriteAds := LIMIT(0,uiWaitBySymbolString_WriteAds,255);
		
		fbADSWrite_WriteAds.IDXGRP := ADSIGRP_SYM_VALBYHND;
			fbADSWrite_WriteAds.IDXOFFS := dwVarHndl_WriteAds;
				fbADSWrite_WriteAds.LEN := uiSizeToWrite_WriteAds;
					fbADSWrite_WriteAds.SRCADDR := ADR(arrBufferWrite_WriteAds);	
						IF byCounterWaitInStep_WriteAds >= 1 THEN fbADSWrite_WriteAds.WRITE := TRUE; END_IF	
	
			IF NOT fbADSWrite_WriteAds.BUSY THEN byCounterWaitInStep_WriteAds := byCounterWaitInStep_WriteAds + 1; END_IF
			
			IF NOT fbADSWrite_WriteAds.BUSY AND NOT fbADSWrite_WriteAds.ERR AND byCounterWaitInStep_WriteAds >= (byStaticValueWaitInStep + uiWaitBySymbolString_WriteAds) THEN 
				fbADSWrite_WriteAds.WRITE := FALSE; 
					iState_WriteAds := 4; 	
						byCounterWaitInStep_WriteAds := 0; 
							uiSizeToWrite_WriteAds := 0;  	
								Lynus_Standards.GVL_Communicator.arrInterfaceInfoValueWriteTo[byReadWriteArrayNumber].bWriteNewValue := FALSE;			
			END_IF

				IF FPErrorWrite_WriteAds.Q OR timTimout_WriteAds.Q THEN iState_WriteAds := 200; END_IF
						
	4://Close Handle
		fbADSWrite_WriteAds.IDXGRP := ADSIGRP_SYM_RELEASEHND;
			fbADSWrite_WriteAds.IDXOFFS := 0;
				fbADSWrite_WriteAds.LEN := SIZEOF(dwVarHndl_WriteAds);
					fbADSWrite_WriteAds.SRCADDR := ADR(dwVarHndl_WriteAds);	
						fbADSWrite_WriteAds.WRITE := TRUE;
							
			IF NOT fbADSWrite_WriteAds.BUSY THEN byCounterWaitInStep_WriteAds := byCounterWaitInStep_WriteAds + 1; END_IF
		
		IF NOT fbADSWrite_WriteAds.BUSY AND NOT fbADSWrite_WriteAds.ERR AND byCounterWaitInStep_WriteAds >= (byStaticValueWaitInStep) THEN 
			fbADSWrite_WriteAds.WRITE := FALSE; 
				Lynus_Standards.GVL_Communicator.arrInterfaceInfoValueWriteTo[byReadWriteArrayNumber].bBusy := FALSE;
					Lynus_Standards.GVL_Communicator.arrInterfaceInfoValueWriteTo[byReadWriteArrayNumber].bErrorWrite := FALSE;
						Lynus_Standards.GVL_Communicator.arrInterfaceInfoValueWriteTo[byReadWriteArrayNumber].sFullSymbolName := '';
							Lynus_Standards.GVL_Communicator.arrInterfaceInfoValueWriteTo[byReadWriteArrayNumber].sSymbolType := '';
								Lynus_Standards.GVL_Communicator.arrInterfaceInfoValueWriteTo[byReadWriteArrayNumber].arrValue := arrValueDefault;	
									Lynus_Standards.GVL_Communicator.arrInterfaceInfoValueWriteTo[byReadWriteArrayNumber].uiSizeArray := 0;
										bError_WriteAds := FALSE;
											uiInternError_WriteAds := 0;
												dwVarHndl_WriteAds := 0; 
													iState_WriteAds := 0; 	
														byCounterWaitInStep_WriteAds := 0;
		END_IF

			IF FPErrorWrite_WriteAds.Q OR timTimout_WriteAds.Q THEN iState_WriteAds := 200; END_IF	
		
	200://Error
		Lynus_Standards.GVL_Communicator.arrInterfaceInfoValueWriteTo[byReadWriteArrayNumber].bErrorWrite := TRUE; Lynus_Standards.GVL_Communicator.arrInterfaceInfoValueWriteTo[byReadWriteArrayNumber].bBusy := FALSE; Lynus_Standards.GVL_Communicator.arrInterfaceInfoValueWriteTo[byReadWriteArrayNumber].bWriteNewValue := FALSE;
			bError_WriteAds := TRUE; fbADSREADWRITE_WriteAds.WRTRD := FALSE; fbADSWrite_WriteAds.WRITE := FALSE; bValueValid_WriteAds := FALSE; Lynus_Standards.GVL_Communicator.arrInterfaceInfoValueWriteTo[byReadWriteArrayNumber].sFullSymbolName := '';
				dwVarHndl_WriteAds := 0; byCounterWaitInStep_WriteAds := 0; byCounterEncodeString_WriteAds := 0; udiDate_WriteAds := 0; uiSizeToWrite_WriteAds := 0; byCounterReceivedValueOK_WriteAds := 0; uiCounterEncodeString_WriteAds := 0;
					uliDate_WriteAds := 0;
		
		iState_WriteAds := 300;
	
	300://Wait in Error
		byCounterWaitInStep_WriteAds := byCounterWaitInStep_WriteAds + 1;
	
			IF byCounterWaitInStep_WriteAds > 10 THEN byCounterWaitInStep_WriteAds := 0; iState_WriteAds := 0; END_IF

END_CASE

//Create Variable Handle
fbADSREADWRITE_WriteAds(
	NETID:= fbNedID.AddrString, 
	PORT:= uiPort, 
	IDXGRP:= ADSIGRP_SYM_HNDBYNAME, 
	IDXOFFS:= 0, 
	WRITELEN:= , 
	READLEN:= SIZEOF(dwVarHndl_WriteAds), 
	SRCADDR:= , 
	DESTADDR:= ADR(dwVarHndl_WriteAds), 
	WRTRD:= , 
	TMOUT:= T#5S, 
	BUSY=> , 
	ERR=> , 
	ERRID=> );

FPErrorReadWrite_WriteAds(CLK:= fbADSREADWRITE_WriteAds.ERR, Q=> );	

//Close Variable Handle	and write Value
fbADSWrite_WriteAds(
	NETID:= fbNedID.AddrString, 
	PORT:= uiPort, 
	IDXGRP:= , 
	IDXOFFS:= , 
	LEN:= , 
	SRCADDR:= , 
	WRITE:= , 
	TMOUT:= T#5S, 
	BUSY=> , 
	ERR=> , 
	ERRID=> );

FPErrorWrite_WriteAds(CLK:= fbADSWrite_WriteAds.ERR, Q=> );
	
//Data read over ADS

CASE iState_ReadAds OF

	-10://Clear Arrays 
		stADSRead_ReadAds := stADSReadDefault_ReadAds;
			stADSReadNew_ReadAds := stADSReadDefault_ReadAds; 
				bError_ReadAds := FALSE; bFirstReadCycleDone_ReadAds := FALSE; bValueIsTheSame_ReadAds := FALSE;
					uiInternError_ReadAds := 0; udiCounterReadBuffer_New_ReadAds := 0; udiActiveNumberOfSymbol_ReadAds := 0; byCounterWaitInStep_ReadAds := 0; 
						udiNumberInProgress_ReadAds := 0; udiRestValueSymbolRead_ReadAds := 0;
							fbBuffer_ReadAds.A_Reset();
	
		//Clear Interface and lengh from each value
		Lynus_Standards.GVL_Communicator.arrInterfaceInfoValueSendTo[byReadWriteArrayNumber].arrValue := arrValueDefault_ReadAds; Lynus_Standards.GVL_Communicator.arrInterfaceInfoValueSendTo[byReadWriteArrayNumber].sSymbolUnit := ''; Lynus_Standards.GVL_Communicator.arrInterfaceInfoValueSendTo[byReadWriteArrayNumber].sFullSymbolName := '';
			Lynus_Standards.GVL_Communicator.arrInterfaceInfoValueSendTo[byReadWriteArrayNumber].sSymbolType := '';	
					
			iState_ReadAds := -9;
	
	-9://Wait from info symbol function	
		IF NOT Lynus_Standards.GVL_Communicator.bBusyInfoAlVariables AND NOT Lynus_Standards.GVL_Communicator.bErrorInfoAlVariables AND Lynus_Standards.GVL_Communicator.bInfoAlVariablesOK AND NOT Lynus_Standards.GVL_Communicator.arrInterfaceInfoValueSendTo[byReadWriteArrayNumber].bErrorSending AND 
			Lynus_Standards.GVL_Communicator.arrInterfaceInfoValueWriteTo[byReadWriteArrayNumber].bSendFunctionOK THEN 
				iState_ReadAds := -8;
		END_IF
			
	-8: //Init
		uiNumberValueSymbolSize_ReadAds := 0; byNumberOfValues_ReadAds_ReadAds := 0; byLenghSymbolName_ReadAds := 0; byValueInTurn_ReadAds := 0; byCounterValue_ReadAds	:= 0;
			uiValueForLoopStart_ReadAds := 0; uiValueForLoopStop_ReadAds := 0; byCounterValueReadOut_ReadAds := 0;
				fbADSREADWRITE_ReadAds.WRTRD := FALSE;	
		arrCounterWriteValueInArray_ReadAds[1] := 0; arrCounterWriteValueInArray_ReadAds[2] := 0; arrCounterWriteValueInArray_ReadAds[3] := 0; arrCounterWriteValueInArray_ReadAds[4] := 0; arrCounterWriteValueInArray_ReadAds[5] := 0;
			arrCounterWriteValueInArray_ReadAds[6] := 0; arrCounterWriteValueInArray_ReadAds[7] := 0; arrCounterWriteValueInArray_ReadAds[8] := 0;
		arrCounterValueSymbolReads_ReadAds[1] := 0;	arrCounterValueSymbolReads_ReadAds[2] := 0; arrCounterValueSymbolReads_ReadAds[3] := 0; arrCounterValueSymbolReads_ReadAds[4] := 0; arrCounterValueSymbolReads_ReadAds[5] := 0;
			arrCounterValueSymbolReads_ReadAds[6] := 0;	arrCounterValueSymbolReads_ReadAds[7] := 0; arrCounterValueSymbolReads_ReadAds[8] := 0; arrCounterValueSymbolReads_ReadAds[9] := 0; arrCounterValueSymbolReads_ReadAds[10] := 0;									
	
		byCounterBufferReq_ReadAds := 0; uiCounterArrayOfString_ReadAds := 0; uiCounterCopyValueFromReqBuffer_ReadAds := 0; udiStartValueReadOutReqBuffer_AdsRead := 0; udiStopValueReadOutReqBuffer_AdsRead := 0;
		
		sStringFloat_ReadAds := ''; iFindPointFloat_ReadAds := 0; iPrecision_ReadAds := 0;
		
		//Copy first 800 default bytes to save resources on small plc's
		MEMCPY(ADR(arrValueAfterRead_ReadAds),ADR(arrValueAfterReadDefault_ReadAds),SIZEOF(arrValueAfterRead_ReadAds));
		
		//Clear lengh from each value
		arrLenghEachValue_ReadAds := arrLenghEachValueDefault_ReadAds;
			
		//Clear array with symbol name and array with the value names
		arrSymbolName_ReadAds := arrSymbolNameDefault_ReadAds;
			arrValueName_ReadAds := arrValueNameDefault_ReadAds;
			
		//Fill numbers of value after each value is read out
		IF udiRestValueSymbolRead_ReadAds = 0 THEN udiRestValueSymbolRead_ReadAds := Lynus_Standards.GVL_Communicator.arrCounterVariableInArray[byReadWriteArrayNumber]; udiStartValueSymbolsRead_ReadAds := 0; udiStopValueSymbolsRead_ReadAds := 0; END_IF 
	
		IF Lynus_Standards.GVL_Communicator.arrCounterVariableInArray[byReadWriteArrayNumber] > 0 THEN iState_ReadAds := -7; byCounterWaitInStep_ReadAds := 0; END_IF  
		
	-7://Prepeare 10 Symbols to read out
		udiStartValueSymbolsRead_ReadAds := udiStopValueSymbolsRead_ReadAds + 1;
			udiStartValueSymbolsRead_ReadAds := LIMIT(1,udiStartValueSymbolsRead_ReadAds,Lynus_Standards.Constants_Communicator.udiArraySizeMarkedSymobls - 9);
				IF udiRestValueSymbolRead_ReadAds > 10 THEN 
					udiStopValueSymbolsRead_ReadAds := udiStopValueSymbolsRead_ReadAds + 10; 
				ELSIF udiRestValueSymbolRead_ReadAds = 10 THEN
					udiStopValueSymbolsRead_ReadAds := udiStopValueSymbolsRead_ReadAds + udiRestValueSymbolRead_ReadAds;
						udiRestValueSymbolRead_ReadAds := 0;
				ELSIF udiRestValueSymbolRead_ReadAds < 10 THEN
					udiStopValueSymbolsRead_ReadAds := udiStopValueSymbolsRead_ReadAds + udiRestValueSymbolRead_ReadAds;
						udiRestValueSymbolRead_ReadAds := 0;
				END_IF
					IF udiRestValueSymbolRead_ReadAds > 10 THEN udiRestValueSymbolRead_ReadAds := udiRestValueSymbolRead_ReadAds - 10; ELSE udiRestValueSymbolRead_ReadAds := udiRestValueSymbolRead_ReadAds; END_IF 	
		
		udiStopValueSymbolsRead_ReadAds := LIMIT(1,udiStopValueSymbolsRead_ReadAds,Lynus_Standards.Constants_Communicator.udiArraySizeMarkedSymobls);
		
			arrCounterValueSymbolReads_ReadAds[1] := udiStartValueSymbolsRead_ReadAds; arrCounterValueSymbolReads_ReadAds[2] := udiStartValueSymbolsRead_ReadAds + 1; arrCounterValueSymbolReads_ReadAds[3] := udiStartValueSymbolsRead_ReadAds + 2;
				arrCounterValueSymbolReads_ReadAds[4] := udiStartValueSymbolsRead_ReadAds + 3; arrCounterValueSymbolReads_ReadAds[5] := udiStartValueSymbolsRead_ReadAds + 4; arrCounterValueSymbolReads_ReadAds[6] := udiStartValueSymbolsRead_ReadAds + 5;
					arrCounterValueSymbolReads_ReadAds[7] := udiStartValueSymbolsRead_ReadAds + 6; arrCounterValueSymbolReads_ReadAds[8] := udiStartValueSymbolsRead_ReadAds + 7; arrCounterValueSymbolReads_ReadAds[9] := udiStartValueSymbolsRead_ReadAds + 8;
						arrCounterValueSymbolReads_ReadAds[10] := udiStartValueSymbolsRead_ReadAds + 9;
			
			udiNumberSizeValues_ReadAds := (udiStopValueSymbolsRead_ReadAds - udiStartValueSymbolsRead_ReadAds + 1);			
			
			FOR byLPClearStructs_ReadAds := 1 TO 10 BY 1 DO
				arrInfoValue_Read_Ads[byLPClearStructs_ReadAds].udiIndexGroup := 0;
				arrInfoValue_Read_Ads[byLPClearStructs_ReadAds].udiIndexOffset := 0;
				arrInfoValue_Read_Ads[byLPClearStructs_ReadAds].udiLength := 0;
			END_FOR
			
				iState_ReadAds := -6;

	-6://Prepeare structs
		arrInfoValue_Read_Ads[1].udiIndexGroup := Lynus_Standards.GVL_Communicator.arrInterfaceInfoAlVariables[byReadWriteArrayNumber,arrCounterValueSymbolReads_ReadAds[1]].udiGroup;
		arrInfoValue_Read_Ads[1].udiIndexOffset := Lynus_Standards.GVL_Communicator.arrInterfaceInfoAlVariables[byReadWriteArrayNumber,arrCounterValueSymbolReads_ReadAds[1]].udiOffset;
		arrInfoValue_Read_Ads[1].udiLength := Lynus_Standards.GVL_Communicator.arrInterfaceInfoAlVariables[byReadWriteArrayNumber,arrCounterValueSymbolReads_ReadAds[1]].udiSize;
			arrInfoValue_Read_Ads[2].udiIndexGroup := Lynus_Standards.GVL_Communicator.arrInterfaceInfoAlVariables[byReadWriteArrayNumber,arrCounterValueSymbolReads_ReadAds[2]].udiGroup;
			arrInfoValue_Read_Ads[2].udiIndexOffset := Lynus_Standards.GVL_Communicator.arrInterfaceInfoAlVariables[byReadWriteArrayNumber,arrCounterValueSymbolReads_ReadAds[2]].udiOffset;
			arrInfoValue_Read_Ads[2].udiLength := Lynus_Standards.GVL_Communicator.arrInterfaceInfoAlVariables[byReadWriteArrayNumber,arrCounterValueSymbolReads_ReadAds[2]].udiSize;
		arrInfoValue_Read_Ads[3].udiIndexGroup := Lynus_Standards.GVL_Communicator.arrInterfaceInfoAlVariables[byReadWriteArrayNumber,arrCounterValueSymbolReads_ReadAds[3]].udiGroup;
		arrInfoValue_Read_Ads[3].udiIndexOffset := Lynus_Standards.GVL_Communicator.arrInterfaceInfoAlVariables[byReadWriteArrayNumber,arrCounterValueSymbolReads_ReadAds[3]].udiOffset;
		arrInfoValue_Read_Ads[3].udiLength := Lynus_Standards.GVL_Communicator.arrInterfaceInfoAlVariables[byReadWriteArrayNumber,arrCounterValueSymbolReads_ReadAds[3]].udiSize;
			arrInfoValue_Read_Ads[4].udiIndexGroup := Lynus_Standards.GVL_Communicator.arrInterfaceInfoAlVariables[byReadWriteArrayNumber,arrCounterValueSymbolReads_ReadAds[4]].udiGroup;
			arrInfoValue_Read_Ads[4].udiIndexOffset := Lynus_Standards.GVL_Communicator.arrInterfaceInfoAlVariables[byReadWriteArrayNumber,arrCounterValueSymbolReads_ReadAds[4]].udiOffset;
			arrInfoValue_Read_Ads[4].udiLength := Lynus_Standards.GVL_Communicator.arrInterfaceInfoAlVariables[byReadWriteArrayNumber,arrCounterValueSymbolReads_ReadAds[4]].udiSize;
		arrInfoValue_Read_Ads[5].udiIndexGroup := Lynus_Standards.GVL_Communicator.arrInterfaceInfoAlVariables[byReadWriteArrayNumber,arrCounterValueSymbolReads_ReadAds[5]].udiGroup;
		arrInfoValue_Read_Ads[5].udiIndexOffset := Lynus_Standards.GVL_Communicator.arrInterfaceInfoAlVariables[byReadWriteArrayNumber,arrCounterValueSymbolReads_ReadAds[5]].udiOffset;
		arrInfoValue_Read_Ads[5].udiLength := Lynus_Standards.GVL_Communicator.arrInterfaceInfoAlVariables[byReadWriteArrayNumber,arrCounterValueSymbolReads_ReadAds[5]].udiSize;
			arrInfoValue_Read_Ads[6].udiIndexGroup := Lynus_Standards.GVL_Communicator.arrInterfaceInfoAlVariables[byReadWriteArrayNumber,arrCounterValueSymbolReads_ReadAds[6]].udiGroup;
			arrInfoValue_Read_Ads[6].udiIndexOffset := Lynus_Standards.GVL_Communicator.arrInterfaceInfoAlVariables[byReadWriteArrayNumber,arrCounterValueSymbolReads_ReadAds[6]].udiOffset;
			arrInfoValue_Read_Ads[6].udiLength := Lynus_Standards.GVL_Communicator.arrInterfaceInfoAlVariables[byReadWriteArrayNumber,arrCounterValueSymbolReads_ReadAds[6]].udiSize;
		arrInfoValue_Read_Ads[7].udiIndexGroup := Lynus_Standards.GVL_Communicator.arrInterfaceInfoAlVariables[byReadWriteArrayNumber,arrCounterValueSymbolReads_ReadAds[7]].udiGroup;
		arrInfoValue_Read_Ads[7].udiIndexOffset := Lynus_Standards.GVL_Communicator.arrInterfaceInfoAlVariables[byReadWriteArrayNumber,arrCounterValueSymbolReads_ReadAds[7]].udiOffset;
		arrInfoValue_Read_Ads[7].udiLength := Lynus_Standards.GVL_Communicator.arrInterfaceInfoAlVariables[byReadWriteArrayNumber,arrCounterValueSymbolReads_ReadAds[7]].udiSize;
			arrInfoValue_Read_Ads[8].udiIndexGroup := Lynus_Standards.GVL_Communicator.arrInterfaceInfoAlVariables[byReadWriteArrayNumber,arrCounterValueSymbolReads_ReadAds[8]].udiGroup;
			arrInfoValue_Read_Ads[8].udiIndexOffset := Lynus_Standards.GVL_Communicator.arrInterfaceInfoAlVariables[byReadWriteArrayNumber,arrCounterValueSymbolReads_ReadAds[8]].udiOffset;
			arrInfoValue_Read_Ads[8].udiLength := Lynus_Standards.GVL_Communicator.arrInterfaceInfoAlVariables[byReadWriteArrayNumber,arrCounterValueSymbolReads_ReadAds[8]].udiSize;
		arrInfoValue_Read_Ads[9].udiIndexGroup := Lynus_Standards.GVL_Communicator.arrInterfaceInfoAlVariables[byReadWriteArrayNumber,arrCounterValueSymbolReads_ReadAds[9]].udiGroup;
		arrInfoValue_Read_Ads[9].udiIndexOffset := Lynus_Standards.GVL_Communicator.arrInterfaceInfoAlVariables[byReadWriteArrayNumber,arrCounterValueSymbolReads_ReadAds[9]].udiOffset;
		arrInfoValue_Read_Ads[9].udiLength := Lynus_Standards.GVL_Communicator.arrInterfaceInfoAlVariables[byReadWriteArrayNumber,arrCounterValueSymbolReads_ReadAds[9]].udiSize;
			arrInfoValue_Read_Ads[10].udiIndexGroup := Lynus_Standards.GVL_Communicator.arrInterfaceInfoAlVariables[byReadWriteArrayNumber,arrCounterValueSymbolReads_ReadAds[10]].udiGroup;
			arrInfoValue_Read_Ads[10].udiIndexOffset := Lynus_Standards.GVL_Communicator.arrInterfaceInfoAlVariables[byReadWriteArrayNumber,arrCounterValueSymbolReads_ReadAds[10]].udiOffset;
			arrInfoValue_Read_Ads[10].udiLength := Lynus_Standards.GVL_Communicator.arrInterfaceInfoAlVariables[byReadWriteArrayNumber,arrCounterValueSymbolReads_ReadAds[10]].udiSize;
	
		MEMCPY(ADR(arrReqValue_ReadAds[1,1]),ADR(arrInfoValue_Read_Ads[1]),SIZEOF(arrInfoValue_Read_Ads[1]));
		MEMCPY(ADR(arrReqValue_ReadAds[2,1]),ADR(arrInfoValue_Read_Ads[2]),SIZEOF(arrInfoValue_Read_Ads[2]));
		MEMCPY(ADR(arrReqValue_ReadAds[3,1]),ADR(arrInfoValue_Read_Ads[3]),SIZEOF(arrInfoValue_Read_Ads[3]));
		MEMCPY(ADR(arrReqValue_ReadAds[4,1]),ADR(arrInfoValue_Read_Ads[4]),SIZEOF(arrInfoValue_Read_Ads[4]));
		MEMCPY(ADR(arrReqValue_ReadAds[5,1]),ADR(arrInfoValue_Read_Ads[5]),SIZEOF(arrInfoValue_Read_Ads[5]));
		MEMCPY(ADR(arrReqValue_ReadAds[6,1]),ADR(arrInfoValue_Read_Ads[6]),SIZEOF(arrInfoValue_Read_Ads[6]));
		MEMCPY(ADR(arrReqValue_ReadAds[7,1]),ADR(arrInfoValue_Read_Ads[7]),SIZEOF(arrInfoValue_Read_Ads[7]));
		MEMCPY(ADR(arrReqValue_ReadAds[8,1]),ADR(arrInfoValue_Read_Ads[8]),SIZEOF(arrInfoValue_Read_Ads[8]));
		MEMCPY(ADR(arrReqValue_ReadAds[9,1]),ADR(arrInfoValue_Read_Ads[9]),SIZEOF(arrInfoValue_Read_Ads[9]));
		MEMCPY(ADR(arrReqValue_ReadAds[10,1]),ADR(arrInfoValue_Read_Ads[10]),SIZEOF(arrInfoValue_Read_Ads[10]));
		
			udiSizeReq_ReadAds := 0;
		
			FOR byLPFillBufferReq_1_ReadAds := 1 TO 10 BY 1 DO
				FOR byLPFillBufferReq_2_ReadAds := 1 TO 12 BY 1 DO
					byCounterBufferReq_ReadAds := LIMIT(1,byCounterBufferReq_ReadAds,120);
						arrBufferReq_ReadAds[byCounterBufferReq_ReadAds] := arrReqValue_ReadAds[byLPFillBufferReq_1_ReadAds,byLPFillBufferReq_2_ReadAds];
							byCounterBufferReq_ReadAds := byCounterBufferReq_ReadAds + 1;
				END_FOR
					udiSizeReq_ReadAds := udiSizeReq_ReadAds + arrInfoValue_Read_Ads[byLPFillBufferReq_1_ReadAds].udiLength;
			END_FOR 
		
		udiSizeReq_ReadAds := udiSizeReq_ReadAds + (udiNumberSizeValues_ReadAds * 4);	
			
		iState_ReadAds := -5;	
			
	-5://Read Values with block mode	
		fbADSREADWRITE_ReadAds.WRITELEN := 12 * udiNumberSizeValues_ReadAds; 	
			fbADSREADWRITE_ReadAds.SRCADDR := ADR(arrBufferReq_ReadAds);
				fbADSREADWRITE_ReadAds.WRTRD := TRUE;	
		
		IF NOT fbADSREADWRITE_ReadAds.BUSY THEN byCounterWaitInStep_ReadAds := byCounterWaitInStep_ReadAds + 1; END_IF  
		
